// TwinCAT 3 PLC project Anker_Modenapark
// ProgramVersion: 3.1.4023.0
// libraries:
//   EfficientIO Communicator, * (EfficientIO)
//   Lynus Energy Basic, * (Lynus AG)
//   Lynus Persistent Data V1, * (Lynus AG)
//   Lynus Standards, * (Lynus AG)
//   Tc2_BABasic, * (Beckhoff Automation GmbH)
//   Tc2_Standard, * (Beckhoff Automation GmbH)
//   Tc2_System, * (Beckhoff Automation GmbH)
//   Tc2_Utilities, * (Beckhoff Automation GmbH)
//   Tc3_IotBase, * (Beckhoff Automation GmbH)
//   Tc3_JsonXml, * (Beckhoff Automation GmbH)
//   Tc3_Module, * (Beckhoff Automation GmbH)
// project tree:
//   / FastTask.TcTTO (not stored), MiddleTask.TcTTO, SlowTask.TcTTO
//   FBs/ FB_Shelly_Pro1PM.TcPOU, FB_Shelly_Pro1PM_Helper.TcPOU, FB_Shelly_Pro1PM_Helper_1.TcPOU (excluded from build), FB_Shelly_Pro1PM_Helper_2.TcPOU (excluded from build), FB_Shelly_Pro1PM_Helper_3.TcPOU (excluded from build), FB_TimeSwitch.TcPOU (not stored), FB_TimeSwitch_V2.TcPOU (not stored)
//   POUs/ prg5532EMS.TcPOU, prg5532Con.TcPOU, prgComEffIO.TcPOU, prg5532Grid.TcPOU, prgPersistent.TcPOU, prgRWEffIO.TcPOU, prgVarEffIO.TcPOU (not stored), prg_SystemTime.TcPOU (not stored)
// real-time tasks:
//   TASK FastTask: cycle T#5ms, priority 19, ADS port 350
//   TASK MiddleTask: cycle T#10ms, priority 20, ADS port 351
//   TASK SlowTask: cycle T#20ms, priority 21, ADS port 352
// I/O:
//   DEVICE Device 1 (Beckhoff CCAT)
//   DEVICE Device 2 (CX-BK)
//     Box 1 (CX-BK)
// variable links:
//   Anker_Modenapark/Anker_Modenapark Instance <-> Device 2 (CX-BK)/Box 1 (CX-BK)
//     MiddleTask Inputs/prg5532Grid.fbGrid.fbKL3403.byStateCH1 <-> Term 3 (KL3403)/Channel 1/State
//     MiddleTask Inputs/prg5532Grid.fbGrid.fbKL3403.byStateCH2 <-> Term 3 (KL3403)/Channel 2/State
//     MiddleTask Inputs/prg5532Grid.fbGrid.fbKL3403.byStateCH3 <-> Term 3 (KL3403)/Channel 3/State
//     MiddleTask Inputs/prg5532Grid.fbGrid.fbKL3403.iDataInCH1 <-> Term 3 (KL3403)/Channel 1/Data In
//     MiddleTask Inputs/prg5532Grid.fbGrid.fbKL3403.iDataInCH2 <-> Term 3 (KL3403)/Channel 2/Data In
//     MiddleTask Inputs/prg5532Grid.fbGrid.fbKL3403.iDataInCH3 <-> Term 3 (KL3403)/Channel 3/Data In
//     MiddleTask Inputs/prg5532Grid.fbKBusState.uiKBusState_OUT <-> Inputs/State
//     MiddleTask Outputs/prg5532EMS.bQ1Switch <-> Term 2 (KL2408)/Channel 1/Output
//     MiddleTask Outputs/prg5532Grid.fbGrid.fbKL3403.byCntrCH1 <-> Term 3 (KL3403)/Channel 1/Ctrl
//     MiddleTask Outputs/prg5532Grid.fbGrid.fbKL3403.byCntrCH2 <-> Term 3 (KL3403)/Channel 2/Ctrl
//     MiddleTask Outputs/prg5532Grid.fbGrid.fbKL3403.byCntrCH3 <-> Term 3 (KL3403)/Channel 3/Ctrl

CONFIGURATION Anker_Modenapark
    RESOURCE PLC ON TwinCAT3
        TASK MiddleTask(INTERVAL := T#10ms, PRIORITY := 20);
        TASK SlowTask(INTERVAL := T#20ms, PRIORITY := 21);
        PROGRAM prgPersistent WITH MiddleTask : prgPersistent;
        PROGRAM prg5532Grid WITH MiddleTask : prg5532Grid;
        PROGRAM prg5532Con WITH MiddleTask : prg5532Con;
        PROGRAM prg5532EMS WITH MiddleTask : prg5532EMS;
        PROGRAM prgComEffIO WITH SlowTask : prgComEffIO;
    END_RESOURCE
END_CONFIGURATION

// ---- POUs/prgPersistent.TcPOU
PROGRAM prgPersistent
VAR
	fbUSV		: FB_WritePersistentData_CX81xx;
END_VAR

fbUSV(
	eSaveModeData:= eUSVSaveMode.eSaveWhenPowerfail, 
	bLoadPersistentDataOk=> , 
	bPowerFailDetect=> , 
	bError=> , 
	bySaveProcess=> , 
	dwStorageLast24h=> , 
	udiErrorCode=> );

END_PROGRAM

// ---- POUs/prg5532Grid.TcPOU
PROGRAM prg5532Grid
VAR
	fbKBusState		: FB_K_Bus_State;
	fbGrid			: FB_EM_Beckhoff_KL3403;
	lrPowerGrid		: LREAL;							//{#lynus.ag#()}
	lrCounterGrid	: LREAL;							//{#lynus.ag#()}
	lrVoltageGridL1	: LREAL;							//{#lynus.ag#()}
	lrVoltageGridL2	: LREAL;							//{#lynus.ag#()}
	lrVoltageGridL3	: LREAL;							//{#lynus.ag#()}
	uint_BusState	: UINT;								//{#lynus.ag#()}
	int_LiveCount:int;
END_VAR

//The mapping of this function must be linked with the K-Bus State in the E/A Part
fbKBusState(	uiKBusState_OUT=> , 
				b_Kbus_notOk=> , 
				word_ErrorCount=> );
				
//The mapping of this function must be linked with the KL3403 in the E/A Part
fbGrid(
	bEnable:= TRUE, 
	bChannel1Invers:= TRUE,					//Invert power data when transformer are mounted upside down
	bChannel2Invers:= TRUE,
	bChannel3Invers:= TRUE,
	uiCurrentTransformerRatioL1:= 400, 		//Transformer ratio on the secondary side
	uiCurrentTransformerRatioL2:= 400, 
	uiCurrentTransformerRatioL3:= 400, 
	uiKBusState_IN:= fbKBusState.uiKBusState_OUT, 
	stDataEMPower=> , 
	stDataEMCounter=> , 
	stDataEMPowerRealTime=> , 
	stDataEMCounterRealTime=> , 
	diNrOfEM_OUT=> );

lrPowerGrid := fbGrid.stDataEMPower.lrPowerTotal;
	lrCounterGrid := fbGrid.stDataEMCounter.lrTotalCounterEnergy_Consumption;
		lrVoltageGridL1 := fbGrid.stDataEMPowerRealTime.lrVoltageL1N;
				lrVoltageGridL2 := fbGrid.stDataEMPowerRealTime.lrVoltageL2N;
					lrVoltageGridL3 := fbGrid.stDataEMPowerRealTime.lrVoltageL3N;


uint_BusState := fbKbusState.uiKBusState_OUT;
int_LiveCount:=int_LiveCount+1;

END_PROGRAM

// ---- POUs/prg5532Con.TcPOU
PROGRAM prg5532Con
VAR
	// Shelly1: 
//	fbShelly1				:	FB_Shelly_Pro1PM;
	lrS1P1Power				:	LREAL;			//{#lynus.ag#()}
	lrS1P1Power_kW			:	LREAL;			//{#lynus.ag#()}
	lrS1P1Voltage			:	LREAL;			//{#lynus.ag#()}
	lrS1P1Energy			:	LREAL;			//{#lynus.ag#()}
	lrS1P1Temperature		:	LREAL;			//{#lynus.ag#()}
	bS1P1On					:	BOOL;			//{#lynus.ag#()}
	bS1P1Off				:	BOOL;			//{#lynus.ag#()}
	bS1P1Switch				:	BOOL;			//{#lynus.ag#()}
	
	// Shelly2: 
//	fbShelly2				:	FB_Shelly_Pro1PM;
	lrS2P1Power				:	LREAL;			//{#lynus.ag#()}
	lrS2P1Power_kW			:	LREAL;			//{#lynus.ag#()}
	lrS2P1Voltage			:	LREAL;			//{#lynus.ag#()}
	lrS2P1Energy			:	LREAL;			//{#lynus.ag#()}
	lrS2P1Temperature		:	LREAL;			//{#lynus.ag#()}
	bS2P1On					:	BOOL;			//{#lynus.ag#()}
	bS2P1Off				:	BOOL;			//{#lynus.ag#()}
	bS2P1Switch				:	BOOL;			//{#lynus.ag#()}
	
	// Shelly3: 
//	fbShelly3				:	FB_Shelly_Pro1PM;
	lrS3P1Power				:	LREAL;			//{#lynus.ag#()}
	lrS3P1Power_kW			:	LREAL;			//{#lynus.ag#()}
	lrS3P1Voltage			:	LREAL;			//{#lynus.ag#()}
	lrS3P1Energy			:	LREAL;			//{#lynus.ag#()}
	lrS3P1Temperature		:	LREAL;			//{#lynus.ag#()}
	bS3P1On					:	BOOL;			//{#lynus.ag#()}
	bS3P1Off				:	BOOL;			//{#lynus.ag#()}
	bS3P1Switch				:	BOOL;			//{#lynus.ag#()}
	
	// Shelly4: 
//	fbShelly4				:	FB_Shelly_Pro1PM;
	lrS4P1Power				:	LREAL;			//{#lynus.ag#()}
	lrS4P1Power_kW			:	LREAL;			//{#lynus.ag#()}
	lrS4P1Voltage			:	LREAL;			//{#lynus.ag#()}
	lrS4P1Energy			:	LREAL;			//{#lynus.ag#()}
	lrS4P1Temperature		:	LREAL;			//{#lynus.ag#()}
	bS4P1On					:	BOOL;			//{#lynus.ag#()}
	bS4P1Off				:	BOOL;			//{#lynus.ag#()}
	bS4P1Switch				:	BOOL;			//{#lynus.ag#()}
	
	// Shelly5: 
//	fbShelly5				:	FB_Shelly_Pro1PM;
	lrS5P1Power				:	LREAL;			//{#lynus.ag#()}
	lrS5P1Power_kW			:	LREAL;			//{#lynus.ag#()}
	lrS5P1Voltage			:	LREAL;			//{#lynus.ag#()}
	lrS5P1Energy			:	LREAL;			//{#lynus.ag#()}
	lrS5P1Temperature		:	LREAL;			//{#lynus.ag#()}
	bS5P1On					:	BOOL;			//{#lynus.ag#()}
	bS5P1Off				:	BOOL;			//{#lynus.ag#()}
	bS5P1Switch				:	BOOL;			//{#lynus.ag#()}
	
	// Other
	lrRemainPower_kW		:	LREAL;			//{#lynus.ag#()}
	// state maschine for GET requests
	str_Array_IPs			: array[1..30] of STRING(15);			//arrays for IPs
	int_State: INT;
	
	int_Multiplier_1 			:INT:=1;								// multilpier received values, =2 when external fuse is on, was at the beginning
	int_Multiplier_2			:INT:=1;								// multilpier received values, =2 when external fuse is on, was at the beginning
	int_Multiplier_3 			:INT:=2;								// multilpier received values, =2 when external fuse is on, was at the beginning
	int_Multiplier_4 			:INT:=2;								// multilpier received values, =2 when external fuse is on, was at the beginning
	int_Multiplier_5 			:INT:=1;								// multilpier received values, =2 when external fuse is on, was at the beginning
	int_TimeoutCounter: ARRAY[1..30] OF INT;	
	int_SuccessCounter: ARRAY[1..30] OF INT;	
	int_ErrorCounter: ARRAY[1..30] OF INT;
	ton_wait: Ton;
	fbShelly				:	ARRAY[1..20] OF FB_Shelly_Pro1PM;
	f_Trig_Busy				:	ARRAY[1..20] OF f_trig;
	m_Error_HTTP: BOOL;							//{#lynus.ag#()}

	mTest: BOOL;
END_VAR

CASE int_State OF
	0: 		// Init State
	
	// define IPs
	str_Array_IPs[1]	:='10.55.32.131';
	str_Array_IPs[2]	:='10.55.32.132';
	str_Array_IPs[3]	:='10.55.32.133';			// bypass aktiv
	str_Array_IPs[4]	:='10.55.32.134';			// bypass aktiv    Getränkekühler RedBull
	str_Array_IPs[5]	:='10.55.32.135';
	str_Array_IPs[6]	:='';
	str_Array_IPs[7]	:='';
	str_Array_IPs[8]	:='';
	str_Array_IPs[9]	:='';
	str_Array_IPs[10]	:='';
	str_Array_IPs[11]	:='';
	str_Array_IPs[12]	:='';
	str_Array_IPs[13]	:='';
	str_Array_IPs[14]	:='';
	fbShelly[1].sHostname:= str_Array_IPs[1];
	fbShelly[2].sHostname:= str_Array_IPs[2];
	fbShelly[3].sHostname:= str_Array_IPs[3];
	fbShelly[4].sHostname:= str_Array_IPs[4];
	fbShelly[5].sHostname:= str_Array_IPs[5];
 
	
	// =2 for the beginning when bypass fuse is on
	int_Multiplier_1:=1;
	int_Multiplier_2:=1;
	int_Multiplier_3:=2;
	int_Multiplier_4:=2;
	int_Multiplier_5:=1;
	
	IF str_Array_IPs[1] <> '' THEN
		int_State :=1;
	END_IF
		
	1: 		// request
	
		fbShelly[int_State].bStart:= TRUE;
		fbShelly[int_State].bOnP1:= bS1P1On;
		fbShelly[int_State].bOffP1:= bS1P1Off;
	
		f_Trig_Busy[int_State](CLK :=fbShelly[int_State].bBusy);
			
		// go to next state
		IF f_Trig_Busy[int_State].Q  AND NOT fbShelly[int_State].bError THEN	
			int_SuccessCounter[int_State]	:= int_SuccessCounter[int_State]+1;
			lrS1P1Power 	:= 	fbShelly[int_State].lrpowerP1 * int_Multiplier_1;
			lrS1P1Energy 	:= 	fbShelly[int_State].lrenergyP1 * int_Multiplier_1;
			lrS1P1Voltage	:=	fbShelly[int_State].lrvoltageP1; 
			lrS1P1Temperature :=fbShelly[int_State].lrTemperatureP1;
			bS1P1Switch		:=	fbShelly[int_State].bStateP1;
		ELSIF  f_Trig_Busy[int_State].Q  AND fbShelly[int_State].bError THEN
			int_ErrorCounter[int_State]	:= int_ErrorCounter[int_State]+1;
		END_IF
		IF 	int_state < 20 AND str_Array_IPs[int_State+1] <> '' AND f_Trig_Busy[int_State].Q  THEN	
			fbShelly[int_State].bStart		:= FALSE;
			int_State := int_State+1;
		ELSIF  (str_Array_IPs[int_State+1] = '' OR int_state > 20) AND f_Trig_Busy[int_State].Q THEN
			fbShelly[int_State].bStart		:= FALSE;
			int_State := 100;			// wait state for new run
		END_IF		
	
	2: 		// request
	
		fbShelly[int_State].bStart:= TRUE;
		fbShelly[int_State].bOnP1:= bS2P1On;
		fbShelly[int_State].bOffP1:= bS2P1Off;
	
		f_Trig_Busy[int_State](CLK :=fbShelly[int_State].bBusy);
			
		// go to next state
		IF f_Trig_Busy[int_State].Q  AND NOT fbShelly[int_State].bError THEN	
			int_SuccessCounter[int_State]	:= int_SuccessCounter[int_State]+1;
			lrS2P1Power 	:= 	fbShelly[int_State].lrpowerP1 * int_Multiplier_2;
			lrS2P1Energy 	:= 	fbShelly[int_State].lrenergyP1 * int_Multiplier_2;
			lrS2P1Temperature :=fbShelly[int_State].lrTemperatureP1;
			lrS2P1Voltage	:=	fbShelly[int_State].lrvoltageP1; 
			bS2P1Switch		:=	fbShelly[int_State].bStateP1;
		ELSIF  f_Trig_Busy[int_State].Q  AND fbShelly[int_State].bError THEN
			int_ErrorCounter[int_State]	:= int_ErrorCounter[int_State]+1;
		END_IF
		IF 	int_state < 20 AND str_Array_IPs[int_State+1] <> '' AND f_Trig_Busy[int_State].Q  THEN	
			fbShelly[int_State].bStart		:= FALSE;
			int_State := int_State+1;
		ELSIF  (str_Array_IPs[int_State+1] = '' OR int_state > 20) AND f_Trig_Busy[int_State].Q THEN
			fbShelly[int_State].bStart		:= FALSE;
			int_State := 100;			// wait state for new run
		END_IF	
		
	3: 		// request
		fbShelly[int_State].bStart:= TRUE;
		fbShelly[int_State].bOnP1:= bS3P1On;
		fbShelly[int_State].bOffP1:= bS3P1Off;
	
		f_Trig_Busy[int_State](CLK :=fbShelly[int_State].bBusy);
			
		// go to next state
		IF f_Trig_Busy[int_State].Q  AND NOT fbShelly[int_State].bError THEN	
			int_SuccessCounter[int_State]	:= int_SuccessCounter[int_State]+1;
			lrS3P1Power 	:= 	fbShelly[int_State].lrpowerP1 * int_Multiplier_3;
			lrS3P1Energy 	:= 	fbShelly[int_State].lrenergyP1 * int_Multiplier_3;
			lrS3P1Temperature :=fbShelly[int_State].lrTemperatureP1;
			lrS3P1Voltage	:=	fbShelly[int_State].lrvoltageP1; 
			bS3P1Switch		:=	fbShelly[int_State].bStateP1;
		ELSIF  f_Trig_Busy[int_State].Q  AND fbShelly[int_State].bError THEN
			int_ErrorCounter[int_State]	:= int_ErrorCounter[int_State]+1;
		END_IF
		IF 	int_state < 20 AND str_Array_IPs[int_State+1] <> '' AND f_Trig_Busy[int_State].Q  THEN	
			fbShelly[int_State].bStart		:= FALSE;
			int_State := int_State+1;
		ELSIF  (str_Array_IPs[int_State+1] = '' OR int_state > 20) AND f_Trig_Busy[int_State].Q THEN
			fbShelly[int_State].bStart		:= FALSE;
			int_State := 100;			// wait state for new run
		END_IF	
	4: 		// request
	
		fbShelly[int_State].bStart:= TRUE;
		fbShelly[int_State].bOnP1:= bS4P1On;
		fbShelly[int_State].bOffP1:= bS4P1Off;
	
		f_Trig_Busy[int_State](CLK :=fbShelly[int_State].bBusy);
		IF f_Trig_Busy[int_State].Q THEN
			mTest:=TRUE;
		END_IF	
		// go to next state
		IF f_Trig_Busy[int_State].Q  AND NOT fbShelly[int_State].bError THEN	
			int_SuccessCounter[int_State]	:= int_SuccessCounter[int_State]+1;
			lrS4P1Power 	:= 	fbShelly[int_State].lrpowerP1 * int_Multiplier_4;
			lrS4P1Energy 	:= 	fbShelly[int_State].lrenergyP1 * int_Multiplier_4;
			lrS4P1Temperature :=fbShelly[int_State].lrTemperatureP1;
			lrS4P1Voltage	:=	fbShelly[int_State].lrvoltageP1; 
			bS4P1Switch		:=	fbShelly[int_State].bStateP1;
		ELSIF  f_Trig_Busy[int_State].Q  AND fbShelly[int_State].bError THEN
			int_ErrorCounter[int_State]	:= int_ErrorCounter[int_State]+1;
		END_IF
		IF 	int_state < 20 AND str_Array_IPs[int_State+1] <> '' AND f_Trig_Busy[int_State].Q  THEN	
			fbShelly[int_State].bStart		:= FALSE;
			int_State := int_State+1;
		ELSIF  (str_Array_IPs[int_State+1] = '' OR int_state > 20) AND f_Trig_Busy[int_State].Q THEN
			fbShelly[int_State].bStart		:= FALSE;
			int_State := 100;			// wait state for new run
		END_IF
		
	5: 		// request
	
		fbShelly[int_State].bStart:= TRUE;
		fbShelly[int_State].bOnP1:= bS5P1On;
		fbShelly[int_State].bOffP1:= bS5P1Off;
	
		f_Trig_Busy[int_State](CLK :=fbShelly[int_State].bBusy);
			
		// go to next state
		IF f_Trig_Busy[int_State].Q  AND NOT fbShelly[int_State].bError THEN	
			int_SuccessCounter[int_State]	:= int_SuccessCounter[int_State]+1;
			lrS5P1Power 	:= 	fbShelly[int_State].lrpowerP1 * int_Multiplier_5;
			lrS5P1Energy 	:= 	fbShelly[int_State].lrenergyP1 * int_Multiplier_5;
			lrS5P1Temperature :=fbShelly[int_State].lrTemperatureP1;
			lrS5P1Voltage	:=	fbShelly[int_State].lrvoltageP1; 
			bS5P1Switch		:=	fbShelly[int_State].bStateP1;
		ELSIF  f_Trig_Busy[int_State].Q  AND fbShelly[int_State].bError THEN
			int_ErrorCounter[int_State]	:= int_ErrorCounter[int_State]+1;
		END_IF
		IF 	int_state < 20 AND str_Array_IPs[int_State+1] <> '' AND f_Trig_Busy[int_State].Q  THEN	
			fbShelly[int_State].bStart		:= FALSE;
			int_State := int_State+1;
		ELSIF  (str_Array_IPs[int_State+1] = '' OR int_state > 20) AND f_Trig_Busy[int_State].Q THEN
			fbShelly[int_State].bStart		:= FALSE;
			int_State := 100;			// wait state for new run
		END_IF	
	
	100:		// wait state
	ton_wait.IN :=TRUE;
	IF ton_wait.Q THEN
		ton_wait.IN :=FALSE;
//		IF NOT fbShelly[1].bError THEN
			int_State := 1;			//// <-- must be 1
//		ELSIF fbShelly[1].bError AND prg_SystemTime.structSystemTime.wHour=4 AND prg_SystemTime.structSystemTime.wMinute>45 THEN
//			int_State := 1;
//		ELSE
//			int_State := 3;
//		END_IF
	END_IF		
END_CASE


// Shelly communication

fbShelly[1](tDelayRequest:= T#0S, );
fbShelly[2](tDelayRequest:= T#0S, );
fbShelly[3](tDelayRequest:= T#0S, );
fbShelly[4](tDelayRequest:= T#0S, );
fbShelly[5](tDelayRequest:= T#0S, );


// wait
ton_wait(PT:=T#3S);


// re-calc to kW
lrS1P1Power_kW := lrS1P1Power / 1000;
	lrS2P1Power_kW := lrS2P1Power / 1000;
		lrS3P1Power_kW := lrS3P1Power / 1000;
			lrS4P1Power_kW := lrS4P1Power / 1000;
				lrS5P1Power_kW := lrS5P1Power / 1000;
				
// Other
lrRemainPower_kW := LIMIT(0, prg5532Grid.lrPowerGrid - (lrS1P1Power_kW + lrS2P1Power_kW + lrS3P1Power_kW + lrS4P1Power_kW + lrS5P1Power_kW), 999999);
	
// on / off commands from EMS

// AC Shelly 1
fbShelly[1].bEnableControl := TRUE;		// prg5532EMS.FB_TimeSwitch_AC.b_Enable;
IF prg5532EMS.FB_TimeSwitch_AC.b_Output_On AND NOT fbShelly[1].bStateP1 THEN
	bS1P1On :=TRUE;
ELSE
	bS1P1On := FALSE;
END_IF
IF NOT prg5532EMS.FB_TimeSwitch_AC.b_Output_On AND fbShelly[1].bStateP1 THEN
	bS1P1Off :=TRUE;
ELSE
	bS1P1Off := FALSE;
END_IF
// Snackvitrine Shelly 2
fbShelly[2].bEnableControl := TRUE;		// prg5532EMS.FB_TimeSwitch_Snack.b_Enable;
IF prg5532EMS.FB_TimeSwitch_Snack.b_Output_On AND NOT fbShelly[2].bStateP1 THEN
	bS2P1On :=TRUE;
ELSE
	bS2P1On := FALSE;
END_IF
IF NOT prg5532EMS.FB_TimeSwitch_Snack.b_Output_On AND fbShelly[2].bStateP1 THEN
	bS2P1Off :=TRUE;
ELSE
	bS2P1Off := FALSE;
END_IF

// Außenbeleuchtung Shelly 5
fbShelly[5].bEnableControl := TRUE;		// prg5532EMS.FB_TimeSwitch_Outside.b_Enable;
IF prg5532EMS.RS_Outsidelight.Q1 AND NOT fbShelly[5].bStateP1 THEN
	bS5P1On :=TRUE;
ELSE
	bS5P1On := FALSE;
END_IF
IF NOT prg5532EMS.RS_Outsidelight.Q1 AND fbShelly[5].bStateP1 THEN
	bS5P1Off :=TRUE;
ELSE
	bS5P1Off := FALSE;
END_IF

// error bit to cloud 

m_Error_HTTP := fbShelly[1].bError OR fbShelly[2].bError OR fbShelly[5].bError;

END_PROGRAM

// ---- FBs/FB_Shelly_Pro1PM.TcPOU
FUNCTION_BLOCK FB_Shelly_Pro1PM
VAR_INPUT
	bStart				: BOOL;
	tDelayRequest		: TIME;				//Timer for delay before start with the next read or write Request
	sHostname			: STRING(255);		//Hostname or IP Adress from the Server
	bOnP1				: BOOL;
	bOffP1				: BOOL;
	bEnableControl		: BOOL;
END_VAR

VAR_OUTPUT
	bValidResult				: BOOL;															//Valid Result received from Server
    bBusy						: BOOL;															//Function is Busy
    bError						: BOOL;															//Error sucess
	bDone						: BOOL;															//True after the decoding from the received Json File
	bConnected					: BOOL;															//Connection to the Server
	hrErrorCode       			: HRESULT;														//Error Result from Http Client
	lrpowerP1					: LREAL;														//Received Value
	lrvoltageP1					: LREAL;														//Received Value
	lrenergyP1					: LREAL;														//Received Value
	lrTemperatureP1				: LREAL;														//Received Value
	bStateP1					: BOOL;
END_VAR

VAR
	fbClient					: FB_IotHttpClient;
	fbHttpGet					: FB_Shelly_Pro1PM_Helper;
	timStartRequest				: TON;															//Timer to Start the Request
	FPStartRequest				: R_TRIG;														//Internal positive Edge
	FPDone						: R_TRIG;														//Internal positive Edge
	FNStart						: F_TRIG;														//Internal negative Edge
	SwitchOnP1					: R_TRIG;
	SwitchOffP1					: R_TRIG;
	rs_Switch_ON: Rs;
	rs_Switch_OFF: RS;
	x: INT;
END_VAR

bError := FALSE;
(*------------------------------------------------------------------------------------Configure HTTP Client------------------------------------------------------------------------------------------------------*)

fbClient.sHostName := sHostname;
fbClient.tConnectionTimeout := T#25S;

IF NOT fbClient.bConfigured THEN 
	fbClient.nHostPort:= 80;
	fbClient.bKeepAlive := TRUE;
	fbClient.tConnectionTimeout := T#25S;
END_IF


//Timer to start the Request
FPStartRequest(CLK:= bStart, Q=> );
timStartRequest(	IN:= fbClient.bConfigured AND bStart AND NOT timStartRequest.Q, 
					PT:= tDelayRequest, 
					Q=> , 
					ET=> );
IF ((timStartRequest.Q AND NOT bBusy) OR (FPStartRequest.Q AND NOT bBusy AND fbClient.bConfigured)) THEN 
	fbHttpGet.bSend := TRUE; 
	x:=x+1;
END_IF

				
//Http Get Function
fbHttpGet(
	lrapowerP1 => lrpowerP1, 
	lrvoltageP1 => lrvoltageP1, 
	lraenergyP1 => lrenergyP1,
	lrTemperatureP1 => lrTemperatureP1,
	bSend:= , 
	fbClient:= fbClient, 
	bBusy=> bBusy, 
	bError=> ,
	sContentS0=> ,
	bStateP1=>bStateP1 );


fbHttpGet.bSend := FALSE;

FPDone(CLK:= bDone, Q=> );

// zum testen ob dadurch die verbindung aufrechtbleibt nach dem schalten 
// --> error geht nicht mehr low!
// IF NOT bError  THEN
	fbClient.Execute();
// ELSE
//	fbClient.Disconnect();
// END_IF

//Error
IF fbHttpGet.bError OR fbClient.bError THEN bError := TRUE; ELSE bError := FALSE; END_IF	
	hrErrorCode := fbClient.hrErrorCode;
	

// Relay Control, Switch P1
SwitchOnP1(CLK:=bOnP1);
rs_Switch_ON(	Set:= SwitchOnP1.Q AND bEnableControl,
				Reset1 := bStateP1);	// OR fbHttpGet.timTimeoutSwitch.Q);
				
IF rs_Switch_ON.Q1 AND bEnableControl THEN
	fbHttpGet.bSetOnP1 := TRUE;
ELSE
	fbHttpGet.bSetOnP1 := FALSE;
END_IF

SwitchOffP1(CLK:=bOffP1);
rs_Switch_OFF(	Set:= SwitchOffP1.Q AND bEnableControl,
				Reset1 := NOT bStateP1);	// OR fbHttpGet.timTimeoutSwitch.Q);
				
IF rs_Switch_OFF.Q1 AND bEnableControl THEN
	fbHttpGet.bSetOffP1 := TRUE;
ELSE
	fbHttpGet.bSetOffP1 := FALSE;
END_IF

END_FUNCTION_BLOCK

// ---- FBs/FB_Shelly_Pro1PM_Helper.TcPOU
FUNCTION_BLOCK FB_Shelly_Pro1PM_Helper
VAR_INPUT
	bSend			: BOOL;
	bSetOnP1		: BOOL;
	bSetOffP1		: BOOL;
END_VAR

VAR_IN_OUT
	fbClient		: FB_IotHttpClient;
END_VAR

VAR_OUTPUT
	bBusy			: BOOL;
	bError			: BOOL;
	bStateP1		: BOOL;
	lrapowerP1		: LREAL;
	lrvoltageP1		: LREAL;
	lraenergyP1		: LREAL;
	lrTemperatureP1	: LREAL;
END_VAR

VAR
	fbRequestSwitch0	: FB_IotHttpRequest;
	fbRequestSwitch1	: FB_IotHttpRequest;
	RisingEdge			: R_TRIG;
	RisingEdgeSetOnP1	: R_TRIG;
	RisingEdgeSetOffP1	: R_TRIG;
	fbJson				: FB_JsonDomParser;
	nState				: UDINT;
	timTimeout			: TON;
	tTimeOut			: TIME := T#2S;
	timTimeoutSwitch	: TON;
	tTimeOutSwitch		: TIME := T#5S;
	bGetContentResult	: BOOL;
	sContentS0			: STRING(511);
	
	bGetJsonResult		: BOOL;
	jsonDoc				: SJsonValue;
	jsonVal				: SJsonValue;
	
	nReqCount			: UDINT;	
	nResCount			: UDINT;
	nValidResCount		: UDINT;
	nErrCount			: UDINT;
	
	fbRequest2         : FB_IotHttpRequest;
	fbRequest3         : FB_IotHttpRequest;
	fbHeader            : FB_IotHttpHeaderFieldMap;
	fbHeader2            : FB_IotHttpHeaderFieldMap;
	
	sRealm	:	STRING(511);
	sPassword :	STRING(511) := ':sh3lly4ankerio2$$';
	snonce	:	STRING(511);
	scnonce	:	STRING(511);
	shash	: STRING(511);
	bhash	: BOOL;
	
	aData	: STRING(511);
	a_ha1	: ARRAY[0..31] OF BYTE;
	str_ha1 : STRING(511);
	str_Toha1   : STRING(511);
	udint_length_string : UDINT;
	
	a_ha2	: ARRAY[0..31] OF BYTE;
	str_ha2 : STRING(511);
	str_Toha2   : STRING(511);
	
	a_response	: ARRAY[0..31] OF BYTE;
	str_response : STRING(511);
	str_Toresponse   : STRING(511);

	str_authorization	: STRING(2048);
	
	sfincontent	: STRING(511);
	int_CountOffWrite: INT;
	int_CountOnWrite: INT;
	str_URI : STRING(50);
	int_Mode: INT;
	ton_Timeout: Ton;
	b_Done: BOOL;
	nState_Old: UDINT;
	int_ErrorCount: INT;
END_VAR

//Timer for Timeout
timTimeout(IN:= (nState = 1 AND bBusy) OR (nState = nState_Old AND bBusy), PT:= tTimeOut, Q=> , ET=> );
	IF timTimeout.Q THEN 
		nState := 0;
		bBusy := FALSE;
		bStateP1 := FALSE;
		lrapowerP1 := 0;
		lrvoltageP1 := 0;
		lraenergyP1 := 0;
		lrTemperatureP1 := 0;		
	END_IF
IF nState<> nState_old THEN
	nState_old := nState;
END_IF	
(*timTimeoutSwitch(IN:= bSetOnP1 OR bSetOffP1, PT:= tTimeOut, Q=> , ET=> );
	IF timTimeoutSwitch.Q THEN 
		bSetOnP1 := FALSE;
		bSetOffP1 := FALSE;
	END_IF
*)
IF bError THEN
	int_ErrorCount := int_ErrorCount+1;
	bError := FALSE;
END_IF

RisingEdge(CLK:= bSend );
RisingEdgeSetOnP1(CLK:= bSetOnP1 );
RisingEdgeSetOffP1(CLK:= bSetOffP1 );

CASE nState OF
	0:	
		IF RisingEdge.Q THEN 
			IF bSetOnP1 AND NOT b_Done THEN 
				// switch on
				str_URI :='/rpc/Switch.Set?id=0&on=true';
				int_Mode := 1;
				b_Done := TRUE;
				bBusy:= TRUE;
				bError:= FALSE;
				nState:= 1;
			ELSIF bSetOffP1 AND NOT b_Done THEN
				// switch off
				str_URI :='/rpc/Switch.Set?id=0&on=false';
				int_Mode := 2;
				b_Done := TRUE;
				bBusy:= TRUE;
				bError:= FALSE;
				nState:= 1;
			ELSIF ((bSetOnP1 OR bSetOffP1) AND  b_Done) OR (NOT bSetOnP1 AND NOT bSetOffP1) THEN
				// read
				str_URI :='/rpc/Switch.GetStatus?id=0';
				int_Mode := 0;
				b_Done := FALSE;
				bBusy:= TRUE;
				bError:= FALSE;
				nState:= 1;
			END_IF
		END_IF
	1:
		IF
			fbRequestSwitch0.SendRequest(sUri:=str_URI, fbClient:=fbClient, eRequestType:=ETcIotHttpRequestType.HTTP_Get, 0, 0, 0) THEN
			nState:= 2;
			nReqCount:= nReqCount+1;
		END_IF
	
	2:
		IF NOT fbRequestSwitch0.bBusy THEN
			bError:= TRUE;
			IF NOT fbRequestSwitch0.bError THEN
				bGetContentResult:= fbRequestSwitch0.GetHeaderField(pValue:= ADR(sContentS0), 
														 nValueSize:= SIZEOF(sContentS0), sField := 'WWW-Authenticate');
				IF fbRequestSwitch0.nStatusCode = 401 THEN
					bGetJsonResult:= FALSE;
						sRealm := sContentS0;
						sRealm := DELETE(sRealm, FIND(sRealm, 'realm') + 7, 0);
						sRealm := DELETE(sRealm, LEN(sRealm), FIND(sRealm, '"'));
						
						snonce := sContentS0;
						snonce := DELETE(snonce, FIND(snonce, 'nonce') + 7, 0);
						snonce := DELETE(snonce, LEN(snonce), FIND(snonce, '"'));
						
						scnonce := 'YmawvYzT';
					
						aData := sRealm;
						
						str_Toha1:=concat('admin:', sRealm);
						str_Toha1:=concat(str_Toha1, sPassword);
		 
						udint_length_string:= len2(ADR(str_Toha1));
						F_GenerateHashValue(E_HashMode.HASH_SHA256,ADR(str_Toha1),udint_length_string,ADR(a_ha1),32);
						
							str_ha1:=concat(byte_to_hexstr(a_ha1[0],2,TRUE),byte_to_hexstr(a_ha1[1],2,TRUE));
							str_ha1:=concat(str_ha1,byte_to_hexstr(a_ha1[2],2,TRUE));
							str_ha1:=concat(str_ha1,byte_to_hexstr(a_ha1[3],2,TRUE));
							str_ha1:=concat(str_ha1,byte_to_hexstr(a_ha1[4],2,TRUE));
							str_ha1:=concat(str_ha1,byte_to_hexstr(a_ha1[5],2,TRUE));
							str_ha1:=concat(str_ha1,byte_to_hexstr(a_ha1[6],2,TRUE));
							str_ha1:=concat(str_ha1,byte_to_hexstr(a_ha1[7],2,TRUE));
							str_ha1:=concat(str_ha1,byte_to_hexstr(a_ha1[8],2,TRUE));
							str_ha1:=concat(str_ha1,byte_to_hexstr(a_ha1[9],2,TRUE));
							str_ha1:=concat(str_ha1,byte_to_hexstr(a_ha1[10],2,TRUE));
							str_ha1:=concat(str_ha1,byte_to_hexstr(a_ha1[11],2,TRUE));
							str_ha1:=concat(str_ha1,byte_to_hexstr(a_ha1[12],2,TRUE));
							str_ha1:=concat(str_ha1,byte_to_hexstr(a_ha1[13],2,TRUE));
							str_ha1:=concat(str_ha1,byte_to_hexstr(a_ha1[14],2,TRUE));
							str_ha1:=concat(str_ha1,byte_to_hexstr(a_ha1[15],2,TRUE));
							str_ha1:=concat(str_ha1,byte_to_hexstr(a_ha1[16],2,TRUE));
							str_ha1:=concat(str_ha1,byte_to_hexstr(a_ha1[17],2,TRUE));
							str_ha1:=concat(str_ha1,byte_to_hexstr(a_ha1[18],2,TRUE));
							str_ha1:=concat(str_ha1,byte_to_hexstr(a_ha1[19],2,TRUE));
							str_ha1:=concat(str_ha1,byte_to_hexstr(a_ha1[20],2,TRUE));
							str_ha1:=concat(str_ha1,byte_to_hexstr(a_ha1[21],2,TRUE));
							str_ha1:=concat(str_ha1,byte_to_hexstr(a_ha1[22],2,TRUE));
							str_ha1:=concat(str_ha1,byte_to_hexstr(a_ha1[23],2,TRUE));
							str_ha1:=concat(str_ha1,byte_to_hexstr(a_ha1[24],2,TRUE));
							str_ha1:=concat(str_ha1,byte_to_hexstr(a_ha1[25],2,TRUE));
							str_ha1:=concat(str_ha1,byte_to_hexstr(a_ha1[26],2,TRUE));
							str_ha1:=concat(str_ha1,byte_to_hexstr(a_ha1[27],2,TRUE));
							str_ha1:=concat(str_ha1,byte_to_hexstr(a_ha1[28],2,TRUE));
							str_ha1:=concat(str_ha1,byte_to_hexstr(a_ha1[29],2,TRUE));
							str_ha1:=concat(str_ha1,byte_to_hexstr(a_ha1[30],2,TRUE));
							str_ha1:=concat(str_ha1,byte_to_hexstr(a_ha1[31],2,TRUE));
						
						str_Toha2:= concat('GET:',str_URI);
				 
						udint_length_string:= len2(ADR(str_Toha2));
						F_GenerateHashValue(E_HashMode.HASH_SHA256,ADR(str_Toha2),udint_length_string,ADR(a_ha2),32);
						
							str_ha2:=concat(byte_to_hexstr(a_ha2[0],2,TRUE),byte_to_hexstr(a_ha2[1],2,TRUE));
							str_ha2:=concat(str_ha2,byte_to_hexstr(a_ha2[2],2,TRUE));
							str_ha2:=concat(str_ha2,byte_to_hexstr(a_ha2[3],2,TRUE));
							str_ha2:=concat(str_ha2,byte_to_hexstr(a_ha2[4],2,TRUE));
							str_ha2:=concat(str_ha2,byte_to_hexstr(a_ha2[5],2,TRUE));
							str_ha2:=concat(str_ha2,byte_to_hexstr(a_ha2[6],2,TRUE));
							str_ha2:=concat(str_ha2,byte_to_hexstr(a_ha2[7],2,TRUE));
							str_ha2:=concat(str_ha2,byte_to_hexstr(a_ha2[8],2,TRUE));
							str_ha2:=concat(str_ha2,byte_to_hexstr(a_ha2[9],2,TRUE));
							str_ha2:=concat(str_ha2,byte_to_hexstr(a_ha2[10],2,TRUE));
							str_ha2:=concat(str_ha2,byte_to_hexstr(a_ha2[11],2,TRUE));
							str_ha2:=concat(str_ha2,byte_to_hexstr(a_ha2[12],2,TRUE));
							str_ha2:=concat(str_ha2,byte_to_hexstr(a_ha2[13],2,TRUE));
							str_ha2:=concat(str_ha2,byte_to_hexstr(a_ha2[14],2,TRUE));
							str_ha2:=concat(str_ha2,byte_to_hexstr(a_ha2[15],2,TRUE));
							str_ha2:=concat(str_ha2,byte_to_hexstr(a_ha2[16],2,TRUE));
							str_ha2:=concat(str_ha2,byte_to_hexstr(a_ha2[17],2,TRUE));
							str_ha2:=concat(str_ha2,byte_to_hexstr(a_ha2[18],2,TRUE));
							str_ha2:=concat(str_ha2,byte_to_hexstr(a_ha2[19],2,TRUE));
							str_ha2:=concat(str_ha2,byte_to_hexstr(a_ha2[20],2,TRUE));
							str_ha2:=concat(str_ha2,byte_to_hexstr(a_ha2[21],2,TRUE));
							str_ha2:=concat(str_ha2,byte_to_hexstr(a_ha2[22],2,TRUE));
							str_ha2:=concat(str_ha2,byte_to_hexstr(a_ha2[23],2,TRUE));
							str_ha2:=concat(str_ha2,byte_to_hexstr(a_ha2[24],2,TRUE));
							str_ha2:=concat(str_ha2,byte_to_hexstr(a_ha2[25],2,TRUE));
							str_ha2:=concat(str_ha2,byte_to_hexstr(a_ha2[26],2,TRUE));
							str_ha2:=concat(str_ha2,byte_to_hexstr(a_ha2[27],2,TRUE));
							str_ha2:=concat(str_ha2,byte_to_hexstr(a_ha2[28],2,TRUE));
							str_ha2:=concat(str_ha2,byte_to_hexstr(a_ha2[29],2,TRUE));
							str_ha2:=concat(str_ha2,byte_to_hexstr(a_ha2[30],2,TRUE));
							str_ha2:=concat(str_ha2,byte_to_hexstr(a_ha2[31],2,TRUE));
							
						// <ha1> + ":" + <nonce> + ":" + <nc> + ":" + <cnonce> + ":" + "auth" + ":" + <ha2>
						
						str_Toresponse:=concat(str_ha1,':');
						str_Toresponse:=concat(str_Toresponse,snonce);
						str_Toresponse:=concat(str_Toresponse,':00000001:');
						str_Toresponse:=concat(str_Toresponse,scnonce);
						str_Toresponse:=concat(str_Toresponse,':');
						str_Toresponse:=concat(str_Toresponse,'auth:');
						str_Toresponse:=concat(str_Toresponse,str_ha2);
						
						udint_length_string:= len2(ADR(str_Toresponse));
						F_GenerateHashValue(E_HashMode.HASH_SHA256,ADR(str_Toresponse),udint_length_string,ADR(a_response),32);
						
							str_response:=concat(byte_to_hexstr(a_response[0],2,TRUE),byte_to_hexstr(a_response[1],2,TRUE));
							str_response:=concat(str_response,byte_to_hexstr(a_response[2],2,TRUE));
							str_response:=concat(str_response,byte_to_hexstr(a_response[3],2,TRUE));
							str_response:=concat(str_response,byte_to_hexstr(a_response[4],2,TRUE));
							str_response:=concat(str_response,byte_to_hexstr(a_response[5],2,TRUE));
							str_response:=concat(str_response,byte_to_hexstr(a_response[6],2,TRUE));
							str_response:=concat(str_response,byte_to_hexstr(a_response[7],2,TRUE));
							str_response:=concat(str_response,byte_to_hexstr(a_response[8],2,TRUE));
							str_response:=concat(str_response,byte_to_hexstr(a_response[9],2,TRUE));
							str_response:=concat(str_response,byte_to_hexstr(a_response[10],2,TRUE));
							str_response:=concat(str_response,byte_to_hexstr(a_response[11],2,TRUE));
							str_response:=concat(str_response,byte_to_hexstr(a_response[12],2,TRUE));
							str_response:=concat(str_response,byte_to_hexstr(a_response[13],2,TRUE));
							str_response:=concat(str_response,byte_to_hexstr(a_response[14],2,TRUE));
							str_response:=concat(str_response,byte_to_hexstr(a_response[15],2,TRUE));
							str_response:=concat(str_response,byte_to_hexstr(a_response[16],2,TRUE));
							str_response:=concat(str_response,byte_to_hexstr(a_response[17],2,TRUE));
							str_response:=concat(str_response,byte_to_hexstr(a_response[18],2,TRUE));
							str_response:=concat(str_response,byte_to_hexstr(a_response[19],2,TRUE));
							str_response:=concat(str_response,byte_to_hexstr(a_response[20],2,TRUE));
							str_response:=concat(str_response,byte_to_hexstr(a_response[21],2,TRUE));
							str_response:=concat(str_response,byte_to_hexstr(a_response[22],2,TRUE));
							str_response:=concat(str_response,byte_to_hexstr(a_response[23],2,TRUE));
							str_response:=concat(str_response,byte_to_hexstr(a_response[24],2,TRUE));
							str_response:=concat(str_response,byte_to_hexstr(a_response[25],2,TRUE));
							str_response:=concat(str_response,byte_to_hexstr(a_response[26],2,TRUE));
							str_response:=concat(str_response,byte_to_hexstr(a_response[27],2,TRUE));
							str_response:=concat(str_response,byte_to_hexstr(a_response[28],2,TRUE));
							str_response:=concat(str_response,byte_to_hexstr(a_response[29],2,TRUE));
							str_response:=concat(str_response,byte_to_hexstr(a_response[30],2,TRUE));
							str_response:=concat(str_response,byte_to_hexstr(a_response[31],2,TRUE));
							
						// "Digest username=\"admin\", realm=\"shellypro4pm-083af27cfbac\", nonce=\"63768368\", uri=\"/rpc/Switch.GetStatus?id=0\", algorithm=\"SHA-256\", qop=auth, nc=00000001, cnonce=\"oKOklSrS\", response=\"d1d59d1e015dee0a3acfc97b20a0fa0ff851b03d79ca00df59ce018a63041468\""
						
						str_authorization:=concat('Digest username="admin", realm="',sRealm);
						str_authorization:=concat(str_authorization,'", nonce="');
						str_authorization:=concat(str_authorization,snonce);
						str_authorization:=concat(str_authorization,'", algorithm="SHA-256", uri="');
						str_authorization:=concat(str_authorization,str_URI);
						str_authorization:=concat(str_authorization,'", qop=auth, nc=00000001, cnonce="');
						str_authorization:=concat(str_authorization,scnonce);
						str_authorization:=concat(str_authorization,'", response="');
						str_authorization:=concat(str_authorization,str_response);
						str_authorization:=concat(str_authorization,'"');
						
						fbHeader.AddField('Authorization', str_authorization, FALSE);
						IF fbRequest2.SendRequest(sUri:= str_URI, fbClient:= fbClient, eRequestType:= ETcIotHttpRequestType.HTTP_Get, 0, 0, fbHeader) THEN
							nState:= 3;
							bBusy:= TRUE;
							bError:= FALSE;
						END_IF
				END_IF
			END_IF
		END_IF
	
	3:
		IF NOT fbRequest2.bBusy THEN
			bError:= TRUE;
			IF int_Mode<>0 THEN
				bError:= FALSE;
			END_IF
			IF NOT fbRequest2.bError THEN		//AND int_Mode=0 				 
				bGetContentResult:= fbRequest2.GetContent(pContent:= ADR(sfincontent), nContentSize:= SIZEOF(sfincontent), bSetNullTermination:= TRUE);
	
				IF fbRequest2.nStatusCode >= 200 AND fbRequest2.nStatusCode < 300 THEN
					bGetJsonResult:= FALSE;
					jsonDoc:= fbRequest2.GetJsonDomContent(fbJson);
					IF jsonDoc <> 0 THEN
						bGetJsonResult:= TRUE;
						IF fbJson.HasMember(jsonDoc, 'output')  THEN
							jsonVal:= fbJson.FindMember(jsonDoc, 'output');
							nValidResCount:= nValidResCount+1;					
							IF fbJson.IsBool(jsonVal) AND (fbJson.GetBool(jsonVal)=TRUE OR fbJson.GetBool(jsonVal)=FALSE) THEN							
								bStateP1:= fbJson.GetBool(jsonVal);									
							END_IF
						END_IF
						IF fbJson.HasMember(jsonDoc, 'apower')  THEN
							jsonVal:= fbJson.FindMember(jsonDoc, 'apower');
							nValidResCount:= nValidResCount+1;
							IF fbJson.IsDouble(jsonVal) AND fbJson.GetDouble(jsonVal)> -3.402823E+38 AND fbJson.GetDouble(jsonVal)< 3.402823E+38 THEN							
								lrapowerP1:= fbJson.GetDouble(jsonVal);									
							END_IF
						END_IF
						IF fbJson.HasMember(jsonDoc, 'voltage')  THEN
							jsonVal:= fbJson.FindMember(jsonDoc, 'voltage');
							nValidResCount:= nValidResCount+1;					
							IF fbJson.IsDouble(jsonVal) AND fbJson.GetDouble(jsonVal)> -3.402823E+38 AND fbJson.GetDouble(jsonVal)< 3.402823E+38 THEN
								lrvoltageP1:= fbJson.GetDouble(jsonVal);									
							END_IF
						END_IF
						IF fbJson.HasMember(jsonDoc, 'temperature')  THEN
							jsonVal:= fbJson.FindMember(jsonDoc, 'temperature');
							 IF fbJson.HasMember(jsonVal, 'tC') AND fbJson.GetDouble(jsonVal)> -3.402823E+38 AND fbJson.GetDouble(jsonVal)< 3.402823E+38 THEN							
								jsonVal:= fbJson.FindMember(jsonVal, 'tC');
								nValidResCount:= nValidResCount+1;					
								IF fbJson.IsDouble(jsonVal) AND fbJson.GetDouble(jsonVal)> -3.402823E+38 AND fbJson.GetDouble(jsonVal)< 3.402823E+38 THEN
									lrTemperatureP1:= fbJson.GetDouble(jsonVal);									
								END_IF
							END_IF
						END_IF
						IF fbJson.HasMember(jsonDoc, 'aenergy')  THEN
							jsonVal:= fbJson.FindMember(jsonDoc, 'aenergy');
							IF fbJson.HasMember(jsonVal, 'total') AND fbJson.GetDouble(jsonVal)> -3.402823E+38 AND fbJson.GetDouble(jsonVal)< 3.402823E+38 THEN							
								jsonVal:= fbJson.FindMember(jsonVal, 'total');
								nValidResCount:= nValidResCount+1;
								IF fbJson.IsDouble(jsonVal) AND fbJson.GetDouble(jsonVal)> -3.402823E+38 AND fbJson.GetDouble(jsonVal)< 3.402823E+38 THEN
									lraenergyP1:= fbJson.GetDouble(jsonVal);
								END_IF
							bError:= FALSE;
							END_IF
						END_IF	
					nResCount:= nResCount+1;			
					END_IF
				END_IF
			END_IF
		nState:= 4;
//		bBusy:= FALSE;
			IF bError THEN
				nErrCount:= nErrCount+1;
			END_IF
		ELSE
			ton_Timeout.IN := TRUE;
			IF ton_Timeout.Q THEN
				nState:= 3;	
				ton_Timeout.IN := FALSE;
			END_IF
		END_IF
	
	
	4:
		ton_Timeout.IN := FALSE;
		nState:= 6;
		
	6:
		bBusy:= FALSE;
		nState:= 0;

	
END_CASE

ton_Timeout(PT := T#5S);

END_FUNCTION_BLOCK

// ---- POUs/prg5532EMS.TcPOU
PROGRAM prg5532EMS
VAR
	//coffee machine relay
	bQ1Switch	AT%Q*	: BOOL;								//{#lynus.ag#()}
	FB_TimeSwitch_Coffee: FB_TimeSwitch_V2;
	FB_TimeSwitch_AC: FB_TimeSwitch_V2;
	FB_TimeSwitch_Snack: FB_TimeSwitch_V2;
	FB_TimeSwitch_RedBull: FB_TimeSwitch_V2;
	FB_TimeSwitch_Outside: FB_TimeSwitch_V2;

	b_Coffee_Manual_On: BOOL;						//{#lynus.ag#()}
	b_Coffee_Manual_Off: BOOL;						//{#lynus.ag#()}
	b_AC_Manual_On: BOOL;							//{#lynus.ag#()}
	b_AC_Manual_Off: BOOL;							//{#lynus.ag#()}
	b_Snack_Manual_On: BOOL;						//{#lynus.ag#()}
	b_Snack_Manual_Off: BOOL;						//{#lynus.ag#()}
	b_Outside_Manual_On: BOOL;						//{#lynus.ag#()}
	b_Outside_Manual_Off: BOOL;						//{#lynus.ag#()}

	fbCalcSunriseSunset   		: FB_CalcSunriseSunset;
	todSunrise            		: TOD;
	todSunset             		: TOD;
	fb_GetTimeZoneInfo	:FB_GetTimeZoneInformation;
	b_firstCycle: BOOL;
	RS_Outsidelight: RS;
	r_trig_on: R_trig;
	r_trig_off: R_trig;
	b_Status_CoffeeMaschine: BOOL;					//{#lynus.ag#()}
END_VAR
VAR PERSISTENT
// opening hours	
	byte_MoFr_Open_Hour		:BYTE;								//{#lynus.ag#()}
	byte_MoFr_Open_Minute	:BYTE;								//{#lynus.ag#()}
	byte_MoFr_Close_Hour	:BYTE;								//{#lynus.ag#()}
	byte_MoFr_Close_Minute	:BYTE;								//{#lynus.ag#()}
	byte_Sa_Open_Hour		:BYTE;								//{#lynus.ag#()}
	byte_Sa_Open_Minute		:BYTE;								//{#lynus.ag#()}
	byte_Sa_Close_Hour		:BYTE;								//{#lynus.ag#()}
	byte_Sa_Close_Minute	:BYTE;								//{#lynus.ag#()}
	byte_So_Open_Hour		:BYTE;								//{#lynus.ag#()}
	byte_So_Open_Minute		:BYTE;								//{#lynus.ag#()}
	byte_So_Close_Hour		:BYTE;								//{#lynus.ag#()}
	byte_So_Close_Minute	:BYTE;								//{#lynus.ag#()}
	
// offset coffeemaschine in hours			
	b_Enable_Control_Coffee		:BOOL;								//{#lynus.ag#()}
	real_Coffee_Offset_Start	:REAL;								//{#lynus.ag#()}
	real_Coffee_Offset_Stop		:REAL;								//{#lynus.ag#()}

// offset AC in hours			
	b_Enable_Control_AC			:BOOL;								//{#lynus.ag#()}
	real_AC_Offset_Start		:REAL;								//{#lynus.ag#()}
	real_AC_Offset_Stop			:REAL;								//{#lynus.ag#()}
	
// offset snack in hours			
	b_Enable_Control_Snack		:BOOL;								//{#lynus.ag#()}
	real_Snack_Offset_Start		:REAL;								//{#lynus.ag#()}
	real_Snack_Offset_Stop		:REAL;								//{#lynus.ag#()}

// offset RedBull Cooler in hours			
	b_Enable_Control_RedBull	:BOOL;								//{#lynus.ag#()}
	real_RedBull_Offset_Start	:REAL;								//{#lynus.ag#()}
	real_RedBull_Offset_Stop	:REAL;								//{#lynus.ag#()}

// offset outside light in hours			
	b_Enable_Control_Outside	:BOOL;								//{#lynus.ag#()}
	real_Outside_Offset_Start	:REAL;								//{#lynus.ag#()}
	real_Outside_Offset_Stop	:REAL;								//{#lynus.ag#()}
END_VAR


FB_TimeSwitch_Coffee(
	b_Enable:= b_Enable_Control_Coffee, 
	b_StatusOn:= NOT bQ1Switch, 
	structSystemTime:=prg_SystemTime.structSystemTime , 
	byte_MoFr_Open_Hour:= byte_MoFr_Open_Hour , 
	byte_MoFr_Open_Minute:= byte_MoFr_Open_Minute, 
	byte_MoFr_Close_Hour:= byte_MoFr_Close_Hour , 
	byte_MoFr_Close_Minute:= byte_MoFr_Close_Minute, 
	byte_Sa_Open_Hour:= byte_Sa_Open_Hour, 
	byte_Sa_Open_Minute:= byte_Sa_Open_Minute , 
	byte_Sa_Close_Hour:= byte_Sa_Close_Hour , 
	byte_Sa_Close_Minute:= byte_Sa_Close_Minute, 
	byte_So_Open_Hour:= byte_So_Open_Hour, 
	byte_So_Open_Minute:= byte_So_Open_Minute, 
	byte_So_Close_Hour:= byte_So_Close_Hour, 
	byte_So_Close_Minute:= byte_So_Close_Minute, 
	real_Offset_Start:= real_Coffee_Offset_Start , 
	real_Offset_Stop:= real_Coffee_Offset_Stop , 
	b_On_Manual:= b_Coffee_Manual_On, 
	b_Off_Manual:= b_Coffee_Manual_Off, 
	b_Output_On=> , 
	b_Error=> );
IF NOT FB_TimeSwitch_Coffee.b_Output_On THEN
	bQ1Switch := TRUE;
ELSIF FB_TimeSwitch_Coffee.b_Output_On THEN
	bQ1Switch := FALSE;
END_IF
b_Status_CoffeeMaschine := NOT bQ1Switch;
	
FB_TimeSwitch_AC(
	b_Enable:= b_Enable_Control_AC, 
	b_StatusOn:= prg5532CON.fbShelly[1].bStateP1, 
	structSystemTime:= prg_SystemTime.structSystemTime , 
	byte_MoFr_Open_Hour:= byte_MoFr_Open_Hour , 
	byte_MoFr_Open_Minute:= byte_MoFr_Open_Minute, 
	byte_MoFr_Close_Hour:= byte_MoFr_Close_Hour , 
	byte_MoFr_Close_Minute:= byte_MoFr_Close_Minute, 
	byte_Sa_Open_Hour:= byte_Sa_Open_Hour, 
	byte_Sa_Open_Minute:= byte_Sa_Open_Minute , 
	byte_Sa_Close_Hour:= byte_Sa_Close_Hour , 
	byte_Sa_Close_Minute:= byte_Sa_Close_Minute, 
	byte_So_Open_Hour:= byte_So_Open_Hour, 
	byte_So_Open_Minute:= byte_So_Open_Minute, 
	byte_So_Close_Hour:= byte_So_Close_Hour, 
	byte_So_Close_Minute:= byte_So_Close_Minute, 
	real_Offset_Start:= real_AC_Offset_Start , 
	real_Offset_Stop:= real_AC_Offset_Stop , 
	b_On_Manual:= b_AC_Manual_On, 
	b_Off_Manual:= b_AC_Manual_Off, 
	b_Output_On=> , 
	b_Error=> );

FB_TimeSwitch_Snack(
	b_Enable:= b_Enable_Control_Snack, 
	b_StatusOn:= prg5532CON.fbShelly[2].bStateP1, 
	structSystemTime:= prg_SystemTime.structSystemTime , 
	byte_MoFr_Open_Hour:= byte_MoFr_Open_Hour , 
	byte_MoFr_Open_Minute:= byte_MoFr_Open_Minute, 
	byte_MoFr_Close_Hour:= byte_MoFr_Close_Hour , 
	byte_MoFr_Close_Minute:= byte_MoFr_Close_Minute, 
	byte_Sa_Open_Hour:= byte_Sa_Open_Hour, 
	byte_Sa_Open_Minute:= byte_Sa_Open_Minute , 
	byte_Sa_Close_Hour:= byte_Sa_Close_Hour , 
	byte_Sa_Close_Minute:= byte_Sa_Close_Minute, 
	byte_So_Open_Hour:= byte_So_Open_Hour, 
	byte_So_Open_Minute:= byte_So_Open_Minute, 
	byte_So_Close_Hour:= byte_So_Close_Hour, 
	byte_So_Close_Minute:= byte_So_Close_Minute, 
	real_Offset_Start:= real_Snack_Offset_Start , 
	real_Offset_Stop:= real_Snack_Offset_Stop , 
	b_On_Manual:= b_Snack_Manual_On, 
	b_Off_Manual:= b_Snack_Manual_Off, 
	b_Output_On=> , 
	b_Error=> );
	
FB_TimeSwitch_Outside(
	b_Enable:= b_Enable_Control_Outside, 
	b_StatusOn:= prg5532CON.fbShelly[5].bStateP1, 
	structSystemTime:= prg_SystemTime.structSystemTime , 
	byte_MoFr_Open_Hour:= byte_MoFr_Open_Hour , 
	byte_MoFr_Open_Minute:= byte_MoFr_Open_Minute, 
	byte_MoFr_Close_Hour:= byte_MoFr_Close_Hour , 
	byte_MoFr_Close_Minute:= byte_MoFr_Close_Minute, 
	byte_Sa_Open_Hour:= byte_Sa_Open_Hour, 
	byte_Sa_Open_Minute:= byte_Sa_Open_Minute , 
	byte_Sa_Close_Hour:= byte_Sa_Close_Hour , 
	byte_Sa_Close_Minute:= byte_Sa_Close_Minute, 
	byte_So_Open_Hour:= byte_So_Open_Hour, 
	byte_So_Open_Minute:= byte_So_Open_Minute, 
	byte_So_Close_Hour:= byte_So_Close_Hour, 
	byte_So_Close_Minute:= byte_So_Close_Minute, 
	real_Offset_Start:= real_Outside_Offset_Start , 
	real_Offset_Stop:= real_Outside_Offset_Stop , 
	b_On_Manual:= b_Outside_Manual_On, 
	b_Off_Manual:= b_Outside_Manual_Off, 
	b_Output_On=> , 
	b_Error=> );
	
// calculate sunset / sunrise
// find out the time details
fb_GetTimeZoneInfo(
	sNetID:= '', 
	bExecute:= prg_SystemTime.structSystemTime.wHour = 4 OR NOT b_firstCycle, 
	tTimeout:= T#5S, 
	bBusy=> , 
	bError=> , 
	nErrID=> , 
	tzID=> , 
	tzInfo=> );
b_firstCycle := TRUE;

fbCalcSunriseSunset(
	fDegreeOfLongitude := 16.3731,   (* Longitude of Vienna *)
	fDegreeOfLatitude := 48.2083,   (* Latitude of Vienna*)
	fReferenceMeridian := SEL( fb_GetTimeZoneInfo.tzID = eTimeZoneID_Daylight ,15,30),  (* Central European Time 15 Winter Timer / 30 Summer Time *)
	dCurrentDate := DT_TO_DATE(SYSTEMTIME_TO_Dt (prg_SystemTime.structSystemTime)),
	todSunrise => todSunrise,
	todSunset => todSunset);

r_trig_on (clk := FB_TimeSwitch_Outside.b_Output_On AND DT_TO_TOD(systemtime_to_dt(prg_SystemTime.structSystemTime))< (todSunrise +  T#1H) );
r_trig_off (clk := NOT FB_TimeSwitch_Outside.b_Output_On);

RS_Outsidelight(	Set := r_trig_on.Q OR ((todSunset - T#2H) =  DT_TO_TOD(systemtime_to_dt(prg_SystemTime.structSystemTime)) AND FB_TimeSwitch_Outside.b_Output_On) OR b_Outside_Manual_On ,
					Reset1 := r_trig_off.Q OR ((todSunrise +  T#1H)= DT_TO_TOD(systemtime_to_dt(prg_SystemTime.structSystemTime))) OR b_Outside_Manual_Off,
					Q1 => );

END_PROGRAM

// ---- POUs/prgComEffIO.TcPOU
PROGRAM prgComEffIO
VAR
	fbCom		: FB_MqttCommunicator;
END_VAR

fbCom(
	bConnect:= TRUE, 
	sUserName:= 'eb1d6961-5914-4eb4-a228-c95326bab078', 
	sUserPassword:= '385e050b-6c7d-4c72-ab76-b82697410544', 
	eSavePositionCertificate:= eSavePositionOnPLC.ePostionHardDisk, 
	bConnected=> , 
	bError=> , 
	hrErrorCode=> , 
	eConnectionState=> , 
	eErrorMessage_Out=> );

prg_SystemTime();

END_PROGRAM

// ---- FBs/FB_Shelly_Pro1PM_Helper_1.TcPOU
FUNCTION_BLOCK FB_Shelly_Pro1PM_Helper_1
VAR_INPUT
	bSend			: BOOL;
	bSetOnP1		: BOOL;
	bSetOffP1		: BOOL;
END_VAR

VAR_IN_OUT
	fbClient		: FB_IotHttpClient;
END_VAR

VAR_OUTPUT
	bBusy			: BOOL;
	bError			: BOOL;
	bStateP1		: BOOL;
	lrapowerP1		: LREAL;
	lrvoltageP1		: LREAL;
	lraenergyP1		: LREAL;
	lrTemperatureP1	: LREAL;
END_VAR

VAR
	fbRequestSwitch0	: FB_IotHttpRequest;
	RisingEdge			: R_TRIG;
	RisingEdgeSetOnP1	: R_TRIG;
	RisingEdgeSetOffP1	: R_TRIG;
	fbJson				: FB_JsonDomParser;
	nState				: UDINT;
	timTimeout			: TON;
	tTimeOut			: TIME := T#30S;
	timTimeoutSwitch	: TON;
	tTimeOutSwitch		: TIME := T#5S;
	bGetContentResult	: BOOL;
	sContentS0			: STRING(511);
	
	bGetJsonResult		: BOOL;
	jsonDoc				: SJsonValue;
	jsonVal				: SJsonValue;
	
	nReqCount			: UDINT;	
	nResCount			: UDINT;
	nValidResCount		: UDINT;
	nErrCount			: UDINT;
	
	fbRequest2         : FB_IotHttpRequest;
	fbHeader            : FB_IotHttpHeaderFieldMap;
	
	sRealm	:	STRING(511);
	sPassword :	STRING(511) := ':sh3lly4ankerio2$$';
	snonce	:	STRING(511);
	scnonce	:	STRING(511);
	shash	: STRING(511);
	bhash	: BOOL;
	
	aData	: STRING(511);
	a_ha1	: ARRAY[0..31] OF BYTE;
	str_ha1 : STRING(511);
	str_Toha1   : STRING(511);
	udint_length_string : UDINT;
	
	a_ha2	: ARRAY[0..31] OF BYTE;
	str_ha2 : STRING(511);
	str_Toha2   : STRING(511);
	
	a_response	: ARRAY[0..31] OF BYTE;
	str_response : STRING(511);
	str_Toresponse   : STRING(511);

	str_authorization	: STRING(2048);
	
	sfincontent	: STRING(511);
END_VAR

//Timer for Timeout
timTimeout(IN:= nState = 1 AND bBusy, PT:= tTimeOut, Q=> , ET=> );
	IF timTimeout.Q THEN 
		nState := 0;
		bBusy := FALSE;
	END_IF
	
timTimeoutSwitch(IN:= bSetOnP1 OR bSetOffP1, PT:= tTimeOut, Q=> , ET=> );
	IF timTimeoutSwitch.Q THEN 
		bSetOnP1 := FALSE;
		bSetOffP1 := FALSE;
	END_IF

RisingEdge(CLK:= bSend );
RisingEdgeSetOnP1(CLK:= bSetOnP1 );
RisingEdgeSetOffP1(CLK:= bSetOffP1 );

CASE nState OF
0:	
	IF RisingEdge.Q THEN 
		IF
			fbRequestSwitch0.SendRequest(sUri:='/rpc/Switch.GetStatus?id=0', fbClient:=fbClient, eRequestType:=ETcIotHttpRequestType.HTTP_Get, 0, 0, 0) THEN
			nState:= 1;
			nReqCount:= nReqCount+1;
			bBusy:= TRUE;
			bError:= FALSE;
		END_IF					
	END_IF
	
	IF RisingEdgeSetOnP1.Q THEN 
		IF
			fbRequestSwitch0.SendRequest(sUri:='/rpc/Switch.Set?id=0&on=true', fbClient:=fbClient, eRequestType:=ETcIotHttpRequestType.HTTP_Get, 0, 0, 0) THEN				
			bSetOnP1 := FALSE;
			nState:= 1;
			bBusy:= TRUE;
			bError:= FALSE;
		END_IF					
	END_IF
	
	IF RisingEdgeSetOffP1.Q THEN 
		IF
			fbRequestSwitch0.SendRequest(sUri:='/rpc/Switch.Set?id=0&on=false', fbClient:=fbClient, eRequestType:=ETcIotHttpRequestType.HTTP_Get, 0, 0, 0) THEN				
			bSetOffP1 := FALSE;
			nState:= 1;
			bBusy:= TRUE;
			bError:= FALSE;
		END_IF					
	END_IF

1:
    IF NOT fbRequestSwitch0.bBusy THEN
        bError:= TRUE;
        IF NOT fbRequestSwitch0.bError THEN
            bGetContentResult:= fbRequestSwitch0.GetHeaderField(pValue:= ADR(sContentS0), 
                                                     nValueSize:= SIZEOF(sContentS0), sField := 'WWW-Authenticate');
            IF fbRequestSwitch0.nStatusCode = 401 THEN
                bGetJsonResult:= FALSE;
					sRealm := sContentS0;
                    sRealm := DELETE(sRealm, FIND(sRealm, 'realm') + 7, 0);
					sRealm := DELETE(sRealm, LEN(sRealm), FIND(sRealm, '"'));
					
					snonce := sContentS0;
					snonce := DELETE(snonce, FIND(snonce, 'nonce') + 7, 0);
					snonce := DELETE(snonce, LEN(snonce), FIND(snonce, '"'));
					
					scnonce := 'YmawvYzT';
				
					aData := sRealm;
					
					str_Toha1:=concat('admin:', sRealm);
    				str_Toha1:=concat(str_Toha1, sPassword);
     
   					udint_length_string:= len2(ADR(str_Toha1));
					F_GenerateHashValue(E_HashMode.HASH_SHA256,ADR(str_Toha1),udint_length_string,ADR(a_ha1),32);
					
						str_ha1:=concat(byte_to_hexstr(a_ha1[0],2,TRUE),byte_to_hexstr(a_ha1[1],2,TRUE));
						str_ha1:=concat(str_ha1,byte_to_hexstr(a_ha1[2],2,TRUE));
						str_ha1:=concat(str_ha1,byte_to_hexstr(a_ha1[3],2,TRUE));
						str_ha1:=concat(str_ha1,byte_to_hexstr(a_ha1[4],2,TRUE));
						str_ha1:=concat(str_ha1,byte_to_hexstr(a_ha1[5],2,TRUE));
						str_ha1:=concat(str_ha1,byte_to_hexstr(a_ha1[6],2,TRUE));
						str_ha1:=concat(str_ha1,byte_to_hexstr(a_ha1[7],2,TRUE));
						str_ha1:=concat(str_ha1,byte_to_hexstr(a_ha1[8],2,TRUE));
						str_ha1:=concat(str_ha1,byte_to_hexstr(a_ha1[9],2,TRUE));
						str_ha1:=concat(str_ha1,byte_to_hexstr(a_ha1[10],2,TRUE));
						str_ha1:=concat(str_ha1,byte_to_hexstr(a_ha1[11],2,TRUE));
						str_ha1:=concat(str_ha1,byte_to_hexstr(a_ha1[12],2,TRUE));
						str_ha1:=concat(str_ha1,byte_to_hexstr(a_ha1[13],2,TRUE));
						str_ha1:=concat(str_ha1,byte_to_hexstr(a_ha1[14],2,TRUE));
						str_ha1:=concat(str_ha1,byte_to_hexstr(a_ha1[15],2,TRUE));
						str_ha1:=concat(str_ha1,byte_to_hexstr(a_ha1[16],2,TRUE));
						str_ha1:=concat(str_ha1,byte_to_hexstr(a_ha1[17],2,TRUE));
						str_ha1:=concat(str_ha1,byte_to_hexstr(a_ha1[18],2,TRUE));
						str_ha1:=concat(str_ha1,byte_to_hexstr(a_ha1[19],2,TRUE));
						str_ha1:=concat(str_ha1,byte_to_hexstr(a_ha1[20],2,TRUE));
						str_ha1:=concat(str_ha1,byte_to_hexstr(a_ha1[21],2,TRUE));
						str_ha1:=concat(str_ha1,byte_to_hexstr(a_ha1[22],2,TRUE));
						str_ha1:=concat(str_ha1,byte_to_hexstr(a_ha1[23],2,TRUE));
						str_ha1:=concat(str_ha1,byte_to_hexstr(a_ha1[24],2,TRUE));
						str_ha1:=concat(str_ha1,byte_to_hexstr(a_ha1[25],2,TRUE));
						str_ha1:=concat(str_ha1,byte_to_hexstr(a_ha1[26],2,TRUE));
						str_ha1:=concat(str_ha1,byte_to_hexstr(a_ha1[27],2,TRUE));
						str_ha1:=concat(str_ha1,byte_to_hexstr(a_ha1[28],2,TRUE));
						str_ha1:=concat(str_ha1,byte_to_hexstr(a_ha1[29],2,TRUE));
						str_ha1:=concat(str_ha1,byte_to_hexstr(a_ha1[30],2,TRUE));
						str_ha1:=concat(str_ha1,byte_to_hexstr(a_ha1[31],2,TRUE));
					
					str_Toha2:='GET:/rpc/Switch.GetStatus?id=0';
     
   					udint_length_string:= len2(ADR(str_Toha2));
					F_GenerateHashValue(E_HashMode.HASH_SHA256,ADR(str_Toha2),udint_length_string,ADR(a_ha2),32);
					
						str_ha2:=concat(byte_to_hexstr(a_ha2[0],2,TRUE),byte_to_hexstr(a_ha2[1],2,TRUE));
						str_ha2:=concat(str_ha2,byte_to_hexstr(a_ha2[2],2,TRUE));
						str_ha2:=concat(str_ha2,byte_to_hexstr(a_ha2[3],2,TRUE));
						str_ha2:=concat(str_ha2,byte_to_hexstr(a_ha2[4],2,TRUE));
						str_ha2:=concat(str_ha2,byte_to_hexstr(a_ha2[5],2,TRUE));
						str_ha2:=concat(str_ha2,byte_to_hexstr(a_ha2[6],2,TRUE));
						str_ha2:=concat(str_ha2,byte_to_hexstr(a_ha2[7],2,TRUE));
						str_ha2:=concat(str_ha2,byte_to_hexstr(a_ha2[8],2,TRUE));
						str_ha2:=concat(str_ha2,byte_to_hexstr(a_ha2[9],2,TRUE));
						str_ha2:=concat(str_ha2,byte_to_hexstr(a_ha2[10],2,TRUE));
						str_ha2:=concat(str_ha2,byte_to_hexstr(a_ha2[11],2,TRUE));
						str_ha2:=concat(str_ha2,byte_to_hexstr(a_ha2[12],2,TRUE));
						str_ha2:=concat(str_ha2,byte_to_hexstr(a_ha2[13],2,TRUE));
						str_ha2:=concat(str_ha2,byte_to_hexstr(a_ha2[14],2,TRUE));
						str_ha2:=concat(str_ha2,byte_to_hexstr(a_ha2[15],2,TRUE));
						str_ha2:=concat(str_ha2,byte_to_hexstr(a_ha2[16],2,TRUE));
						str_ha2:=concat(str_ha2,byte_to_hexstr(a_ha2[17],2,TRUE));
						str_ha2:=concat(str_ha2,byte_to_hexstr(a_ha2[18],2,TRUE));
						str_ha2:=concat(str_ha2,byte_to_hexstr(a_ha2[19],2,TRUE));
						str_ha2:=concat(str_ha2,byte_to_hexstr(a_ha2[20],2,TRUE));
						str_ha2:=concat(str_ha2,byte_to_hexstr(a_ha2[21],2,TRUE));
						str_ha2:=concat(str_ha2,byte_to_hexstr(a_ha2[22],2,TRUE));
						str_ha2:=concat(str_ha2,byte_to_hexstr(a_ha2[23],2,TRUE));
						str_ha2:=concat(str_ha2,byte_to_hexstr(a_ha2[24],2,TRUE));
						str_ha2:=concat(str_ha2,byte_to_hexstr(a_ha2[25],2,TRUE));
						str_ha2:=concat(str_ha2,byte_to_hexstr(a_ha2[26],2,TRUE));
						str_ha2:=concat(str_ha2,byte_to_hexstr(a_ha2[27],2,TRUE));
						str_ha2:=concat(str_ha2,byte_to_hexstr(a_ha2[28],2,TRUE));
						str_ha2:=concat(str_ha2,byte_to_hexstr(a_ha2[29],2,TRUE));
						str_ha2:=concat(str_ha2,byte_to_hexstr(a_ha2[30],2,TRUE));
						str_ha2:=concat(str_ha2,byte_to_hexstr(a_ha2[31],2,TRUE));
						
					// <ha1> + ":" + <nonce> + ":" + <nc> + ":" + <cnonce> + ":" + "auth" + ":" + <ha2>
					
					str_Toresponse:=concat(str_ha1,':');
					str_Toresponse:=concat(str_Toresponse,snonce);
					str_Toresponse:=concat(str_Toresponse,':00000001:');
					str_Toresponse:=concat(str_Toresponse,scnonce);
					str_Toresponse:=concat(str_Toresponse,':');
					str_Toresponse:=concat(str_Toresponse,'auth:');
					str_Toresponse:=concat(str_Toresponse,str_ha2);
					
					udint_length_string:= len2(ADR(str_Toresponse));
					F_GenerateHashValue(E_HashMode.HASH_SHA256,ADR(str_Toresponse),udint_length_string,ADR(a_response),32);
					
						str_response:=concat(byte_to_hexstr(a_response[0],2,TRUE),byte_to_hexstr(a_response[1],2,TRUE));
						str_response:=concat(str_response,byte_to_hexstr(a_response[2],2,TRUE));
						str_response:=concat(str_response,byte_to_hexstr(a_response[3],2,TRUE));
						str_response:=concat(str_response,byte_to_hexstr(a_response[4],2,TRUE));
						str_response:=concat(str_response,byte_to_hexstr(a_response[5],2,TRUE));
						str_response:=concat(str_response,byte_to_hexstr(a_response[6],2,TRUE));
						str_response:=concat(str_response,byte_to_hexstr(a_response[7],2,TRUE));
						str_response:=concat(str_response,byte_to_hexstr(a_response[8],2,TRUE));
						str_response:=concat(str_response,byte_to_hexstr(a_response[9],2,TRUE));
						str_response:=concat(str_response,byte_to_hexstr(a_response[10],2,TRUE));
						str_response:=concat(str_response,byte_to_hexstr(a_response[11],2,TRUE));
						str_response:=concat(str_response,byte_to_hexstr(a_response[12],2,TRUE));
						str_response:=concat(str_response,byte_to_hexstr(a_response[13],2,TRUE));
						str_response:=concat(str_response,byte_to_hexstr(a_response[14],2,TRUE));
						str_response:=concat(str_response,byte_to_hexstr(a_response[15],2,TRUE));
						str_response:=concat(str_response,byte_to_hexstr(a_response[16],2,TRUE));
						str_response:=concat(str_response,byte_to_hexstr(a_response[17],2,TRUE));
						str_response:=concat(str_response,byte_to_hexstr(a_response[18],2,TRUE));
						str_response:=concat(str_response,byte_to_hexstr(a_response[19],2,TRUE));
						str_response:=concat(str_response,byte_to_hexstr(a_response[20],2,TRUE));
						str_response:=concat(str_response,byte_to_hexstr(a_response[21],2,TRUE));
						str_response:=concat(str_response,byte_to_hexstr(a_response[22],2,TRUE));
						str_response:=concat(str_response,byte_to_hexstr(a_response[23],2,TRUE));
						str_response:=concat(str_response,byte_to_hexstr(a_response[24],2,TRUE));
						str_response:=concat(str_response,byte_to_hexstr(a_response[25],2,TRUE));
						str_response:=concat(str_response,byte_to_hexstr(a_response[26],2,TRUE));
						str_response:=concat(str_response,byte_to_hexstr(a_response[27],2,TRUE));
						str_response:=concat(str_response,byte_to_hexstr(a_response[28],2,TRUE));
						str_response:=concat(str_response,byte_to_hexstr(a_response[29],2,TRUE));
						str_response:=concat(str_response,byte_to_hexstr(a_response[30],2,TRUE));
						str_response:=concat(str_response,byte_to_hexstr(a_response[31],2,TRUE));
						
					// "Digest username=\"admin\", realm=\"shellypro4pm-083af27cfbac\", nonce=\"63768368\", uri=\"/rpc/Switch.GetStatus?id=0\", algorithm=\"SHA-256\", qop=auth, nc=00000001, cnonce=\"oKOklSrS\", response=\"d1d59d1e015dee0a3acfc97b20a0fa0ff851b03d79ca00df59ce018a63041468\""
					
					str_authorization:=concat('Digest username="admin", realm="',sRealm);
					str_authorization:=concat(str_authorization,'", nonce="');
					str_authorization:=concat(str_authorization,snonce);
					str_authorization:=concat(str_authorization,'", algorithm="SHA-256", uri="/rpc/Switch.GetStatus?id=0", qop=auth, nc=00000001, cnonce="');
					str_authorization:=concat(str_authorization,scnonce);
					str_authorization:=concat(str_authorization,'", response="');
					str_authorization:=concat(str_authorization,str_response);
					str_authorization:=concat(str_authorization,'"');
					
					fbHeader.AddField('Authorization', str_authorization, FALSE);
					IF fbRequest2.SendRequest(sUri:= '/rpc/Switch.GetStatus?id=0', fbClient:= fbClient, eRequestType:= ETcIotHttpRequestType.HTTP_Get, 0, 0, fbHeader) THEN
						nState:= 2;
						bBusy:= TRUE;
						bError:= FALSE;
					END_IF
			END_IF
		END_IF
	END_IF


2:
	IF NOT fbRequest2.bBusy THEN
		bError:= TRUE;
		
		IF NOT fbRequest2.bError THEN				 
			bGetContentResult:= fbRequest2.GetContent(pContent:= ADR(sfincontent), nContentSize:= SIZEOF(sfincontent), bSetNullTermination:= TRUE);

			IF fbRequest2.nStatusCode >= 200 AND fbRequest2.nStatusCode < 300 THEN
				bGetJsonResult:= FALSE;
				jsonDoc:= fbRequest2.GetJsonDomContent(fbJson);
				IF jsonDoc <> 0 THEN
					bGetJsonResult:= TRUE;
					IF fbJson.HasMember(jsonDoc, 'output')  THEN
						jsonVal:= fbJson.FindMember(jsonDoc, 'output');
						nValidResCount:= nValidResCount+1;					
						IF fbJson.IsBool(jsonVal) AND (fbJson.GetBool(jsonVal)=TRUE OR fbJson.GetBool(jsonVal)=FALSE) THEN							
							bStateP1:= fbJson.GetBool(jsonVal);									
						END_IF
					END_IF
					IF fbJson.HasMember(jsonDoc, 'apower')  THEN
						jsonVal:= fbJson.FindMember(jsonDoc, 'apower');
						nValidResCount:= nValidResCount+1;
						IF fbJson.IsDouble(jsonVal) AND fbJson.GetDouble(jsonVal)> -3.402823E+38 AND fbJson.GetDouble(jsonVal)< 3.402823E+38 THEN							
							lrapowerP1:= fbJson.GetDouble(jsonVal);									
						END_IF
					END_IF
					IF fbJson.HasMember(jsonDoc, 'voltage')  THEN
						jsonVal:= fbJson.FindMember(jsonDoc, 'voltage');
						nValidResCount:= nValidResCount+1;					
						IF fbJson.IsDouble(jsonVal) AND fbJson.GetDouble(jsonVal)> -3.402823E+38 AND fbJson.GetDouble(jsonVal)< 3.402823E+38 THEN
							lrvoltageP1:= fbJson.GetDouble(jsonVal);									
						END_IF
					END_IF
					IF fbJson.HasMember(jsonDoc, 'temperature')  THEN
						jsonVal:= fbJson.FindMember(jsonDoc, 'temperature');
						 IF fbJson.HasMember(jsonVal, 'tC') AND fbJson.GetDouble(jsonVal)> -3.402823E+38 AND fbJson.GetDouble(jsonVal)< 3.402823E+38 THEN							
                            jsonVal:= fbJson.FindMember(jsonVal, 'tC');
							nValidResCount:= nValidResCount+1;					
							IF fbJson.IsDouble(jsonVal) AND fbJson.GetDouble(jsonVal)> -3.402823E+38 AND fbJson.GetDouble(jsonVal)< 3.402823E+38 THEN
								lrTemperatureP1:= fbJson.GetDouble(jsonVal);									
							END_IF
						END_IF
					END_IF
					IF fbJson.HasMember(jsonDoc, 'aenergy')  THEN
						jsonVal:= fbJson.FindMember(jsonDoc, 'aenergy');
                        IF fbJson.HasMember(jsonVal, 'total') AND fbJson.GetDouble(jsonVal)> -3.402823E+38 AND fbJson.GetDouble(jsonVal)< 3.402823E+38 THEN							
                            jsonVal:= fbJson.FindMember(jsonVal, 'total');
                            nValidResCount:= nValidResCount+1;
                            IF fbJson.IsDouble(jsonVal) AND fbJson.GetDouble(jsonVal)> -3.402823E+38 AND fbJson.GetDouble(jsonVal)< 3.402823E+38 THEN
                                lraenergyP1:= fbJson.GetDouble(jsonVal);
                            END_IF
						bError:= FALSE;
						END_IF
					END_IF	

				nResCount:= nResCount+1;			
				END_IF
			END_IF
		END_IF
		
	nState:= 0;
	bBusy:= FALSE;
		IF bError THEN
			nErrCount:= nErrCount+1;
		END_IF
	END_IF
	
END_CASE

END_FUNCTION_BLOCK

// ---- FBs/FB_Shelly_Pro1PM_Helper_2.TcPOU
FUNCTION_BLOCK FB_Shelly_Pro1PM_Helper_2
VAR_INPUT
	bSend			: BOOL;
	bSetOnP1		: BOOL;
	bSetOffP1		: BOOL;
END_VAR

VAR_IN_OUT
	fbClient		: FB_IotHttpClient;
END_VAR

VAR_OUTPUT
	bBusy			: BOOL;
	bError			: BOOL;
	bStateP1		: BOOL;
	lrapowerP1		: LREAL;
	lrvoltageP1		: LREAL;
	lraenergyP1		: LREAL;
	lrTemperatureP1	: LREAL;
END_VAR

VAR
	fbRequestSwitch0	: FB_IotHttpRequest;
	RisingEdge			: R_TRIG;
	RisingEdgeSetOnP1	: R_TRIG;
	RisingEdgeSetOffP1	: R_TRIG;
	fbJson				: FB_JsonDomParser;
	nState				: UDINT;
	timTimeout			: TON;
	tTimeOut			: TIME := T#30S;
	timTimeoutSwitch	: TON;
	tTimeOutSwitch		: TIME := T#5S;
	bGetContentResult	: BOOL;
	sContentS0			: STRING(511);
	
	bGetJsonResult		: BOOL;
	jsonDoc				: SJsonValue;
	jsonVal				: SJsonValue;
	
	nReqCount			: UDINT;	
	nResCount			: UDINT;
	nValidResCount		: UDINT;
	nErrCount			: UDINT;
	
	fbRequest2         : FB_IotHttpRequest;
	fbRequest3         : FB_IotHttpRequest;
	fbHeader            : FB_IotHttpHeaderFieldMap;
	
	sRealm	:	STRING(511);
	sPassword :	STRING(511) := ':sh3lly4ankerio2$$';
	snonce	:	STRING(511);
	scnonce	:	STRING(511);
	shash	: STRING(511);
	bhash	: BOOL;
	
	aData	: STRING(511);
	a_ha1	: ARRAY[0..31] OF BYTE;
	str_ha1 : STRING(511);
	str_Toha1   : STRING(511);
	udint_length_string : UDINT;
	
	a_ha2	: ARRAY[0..31] OF BYTE;
	str_ha2 : STRING(511);
	str_Toha2   : STRING(511);
	
	a_response	: ARRAY[0..31] OF BYTE;
	str_response : STRING(511);
	str_Toresponse   : STRING(511);

	str_authorization	: STRING(2048);
	
	sfincontent	: STRING(511);
	int_CountOffWrite: INT;
	int_CountOnWrite: INT;
END_VAR

//Timer for Timeout
timTimeout(IN:= nState = 1 AND bBusy, PT:= tTimeOut, Q=> , ET=> );
	IF timTimeout.Q THEN 
		nState := 0;
		bBusy := FALSE;
	END_IF
	
timTimeoutSwitch(IN:= bSetOnP1 OR bSetOffP1, PT:= tTimeOut, Q=> , ET=> );
	IF timTimeoutSwitch.Q THEN 
		bSetOnP1 := FALSE;
		bSetOffP1 := FALSE;
	END_IF

RisingEdge(CLK:= bSend );
RisingEdgeSetOnP1(CLK:= bSetOnP1 );
RisingEdgeSetOffP1(CLK:= bSetOffP1 );

CASE nState OF
	0:	
		IF RisingEdge.Q THEN 
			IF
				fbRequestSwitch0.SendRequest(sUri:='/rpc/Switch.GetStatus?id=0', fbClient:=fbClient, eRequestType:=ETcIotHttpRequestType.HTTP_Get, 0, 0, 0) THEN
				nState:= 1;
				nReqCount:= nReqCount+1;
				bBusy:= TRUE;
				bError:= FALSE;
			END_IF					
		END_IF
	1:
		IF NOT fbRequestSwitch0.bBusy THEN
			bError:= TRUE;
			IF NOT fbRequestSwitch0.bError THEN
				bGetContentResult:= fbRequestSwitch0.GetHeaderField(pValue:= ADR(sContentS0), 
														 nValueSize:= SIZEOF(sContentS0), sField := 'WWW-Authenticate');
				IF fbRequestSwitch0.nStatusCode = 401 THEN
					bGetJsonResult:= FALSE;
						sRealm := sContentS0;
						sRealm := DELETE(sRealm, FIND(sRealm, 'realm') + 7, 0);
						sRealm := DELETE(sRealm, LEN(sRealm), FIND(sRealm, '"'));
						
						snonce := sContentS0;
						snonce := DELETE(snonce, FIND(snonce, 'nonce') + 7, 0);
						snonce := DELETE(snonce, LEN(snonce), FIND(snonce, '"'));
						
						scnonce := 'YmawvYzT';
					
						aData := sRealm;
						
						str_Toha1:=concat('admin:', sRealm);
						str_Toha1:=concat(str_Toha1, sPassword);
		 
						udint_length_string:= len2(ADR(str_Toha1));
						F_GenerateHashValue(E_HashMode.HASH_SHA256,ADR(str_Toha1),udint_length_string,ADR(a_ha1),32);
						
							str_ha1:=concat(byte_to_hexstr(a_ha1[0],2,TRUE),byte_to_hexstr(a_ha1[1],2,TRUE));
							str_ha1:=concat(str_ha1,byte_to_hexstr(a_ha1[2],2,TRUE));
							str_ha1:=concat(str_ha1,byte_to_hexstr(a_ha1[3],2,TRUE));
							str_ha1:=concat(str_ha1,byte_to_hexstr(a_ha1[4],2,TRUE));
							str_ha1:=concat(str_ha1,byte_to_hexstr(a_ha1[5],2,TRUE));
							str_ha1:=concat(str_ha1,byte_to_hexstr(a_ha1[6],2,TRUE));
							str_ha1:=concat(str_ha1,byte_to_hexstr(a_ha1[7],2,TRUE));
							str_ha1:=concat(str_ha1,byte_to_hexstr(a_ha1[8],2,TRUE));
							str_ha1:=concat(str_ha1,byte_to_hexstr(a_ha1[9],2,TRUE));
							str_ha1:=concat(str_ha1,byte_to_hexstr(a_ha1[10],2,TRUE));
							str_ha1:=concat(str_ha1,byte_to_hexstr(a_ha1[11],2,TRUE));
							str_ha1:=concat(str_ha1,byte_to_hexstr(a_ha1[12],2,TRUE));
							str_ha1:=concat(str_ha1,byte_to_hexstr(a_ha1[13],2,TRUE));
							str_ha1:=concat(str_ha1,byte_to_hexstr(a_ha1[14],2,TRUE));
							str_ha1:=concat(str_ha1,byte_to_hexstr(a_ha1[15],2,TRUE));
							str_ha1:=concat(str_ha1,byte_to_hexstr(a_ha1[16],2,TRUE));
							str_ha1:=concat(str_ha1,byte_to_hexstr(a_ha1[17],2,TRUE));
							str_ha1:=concat(str_ha1,byte_to_hexstr(a_ha1[18],2,TRUE));
							str_ha1:=concat(str_ha1,byte_to_hexstr(a_ha1[19],2,TRUE));
							str_ha1:=concat(str_ha1,byte_to_hexstr(a_ha1[20],2,TRUE));
							str_ha1:=concat(str_ha1,byte_to_hexstr(a_ha1[21],2,TRUE));
							str_ha1:=concat(str_ha1,byte_to_hexstr(a_ha1[22],2,TRUE));
							str_ha1:=concat(str_ha1,byte_to_hexstr(a_ha1[23],2,TRUE));
							str_ha1:=concat(str_ha1,byte_to_hexstr(a_ha1[24],2,TRUE));
							str_ha1:=concat(str_ha1,byte_to_hexstr(a_ha1[25],2,TRUE));
							str_ha1:=concat(str_ha1,byte_to_hexstr(a_ha1[26],2,TRUE));
							str_ha1:=concat(str_ha1,byte_to_hexstr(a_ha1[27],2,TRUE));
							str_ha1:=concat(str_ha1,byte_to_hexstr(a_ha1[28],2,TRUE));
							str_ha1:=concat(str_ha1,byte_to_hexstr(a_ha1[29],2,TRUE));
							str_ha1:=concat(str_ha1,byte_to_hexstr(a_ha1[30],2,TRUE));
							str_ha1:=concat(str_ha1,byte_to_hexstr(a_ha1[31],2,TRUE));
						
						str_Toha2:='GET:/rpc/Switch.GetStatus?id=0';
		 
						udint_length_string:= len2(ADR(str_Toha2));
						F_GenerateHashValue(E_HashMode.HASH_SHA256,ADR(str_Toha2),udint_length_string,ADR(a_ha2),32);
						
							str_ha2:=concat(byte_to_hexstr(a_ha2[0],2,TRUE),byte_to_hexstr(a_ha2[1],2,TRUE));
							str_ha2:=concat(str_ha2,byte_to_hexstr(a_ha2[2],2,TRUE));
							str_ha2:=concat(str_ha2,byte_to_hexstr(a_ha2[3],2,TRUE));
							str_ha2:=concat(str_ha2,byte_to_hexstr(a_ha2[4],2,TRUE));
							str_ha2:=concat(str_ha2,byte_to_hexstr(a_ha2[5],2,TRUE));
							str_ha2:=concat(str_ha2,byte_to_hexstr(a_ha2[6],2,TRUE));
							str_ha2:=concat(str_ha2,byte_to_hexstr(a_ha2[7],2,TRUE));
							str_ha2:=concat(str_ha2,byte_to_hexstr(a_ha2[8],2,TRUE));
							str_ha2:=concat(str_ha2,byte_to_hexstr(a_ha2[9],2,TRUE));
							str_ha2:=concat(str_ha2,byte_to_hexstr(a_ha2[10],2,TRUE));
							str_ha2:=concat(str_ha2,byte_to_hexstr(a_ha2[11],2,TRUE));
							str_ha2:=concat(str_ha2,byte_to_hexstr(a_ha2[12],2,TRUE));
							str_ha2:=concat(str_ha2,byte_to_hexstr(a_ha2[13],2,TRUE));
							str_ha2:=concat(str_ha2,byte_to_hexstr(a_ha2[14],2,TRUE));
							str_ha2:=concat(str_ha2,byte_to_hexstr(a_ha2[15],2,TRUE));
							str_ha2:=concat(str_ha2,byte_to_hexstr(a_ha2[16],2,TRUE));
							str_ha2:=concat(str_ha2,byte_to_hexstr(a_ha2[17],2,TRUE));
							str_ha2:=concat(str_ha2,byte_to_hexstr(a_ha2[18],2,TRUE));
							str_ha2:=concat(str_ha2,byte_to_hexstr(a_ha2[19],2,TRUE));
							str_ha2:=concat(str_ha2,byte_to_hexstr(a_ha2[20],2,TRUE));
							str_ha2:=concat(str_ha2,byte_to_hexstr(a_ha2[21],2,TRUE));
							str_ha2:=concat(str_ha2,byte_to_hexstr(a_ha2[22],2,TRUE));
							str_ha2:=concat(str_ha2,byte_to_hexstr(a_ha2[23],2,TRUE));
							str_ha2:=concat(str_ha2,byte_to_hexstr(a_ha2[24],2,TRUE));
							str_ha2:=concat(str_ha2,byte_to_hexstr(a_ha2[25],2,TRUE));
							str_ha2:=concat(str_ha2,byte_to_hexstr(a_ha2[26],2,TRUE));
							str_ha2:=concat(str_ha2,byte_to_hexstr(a_ha2[27],2,TRUE));
							str_ha2:=concat(str_ha2,byte_to_hexstr(a_ha2[28],2,TRUE));
							str_ha2:=concat(str_ha2,byte_to_hexstr(a_ha2[29],2,TRUE));
							str_ha2:=concat(str_ha2,byte_to_hexstr(a_ha2[30],2,TRUE));
							str_ha2:=concat(str_ha2,byte_to_hexstr(a_ha2[31],2,TRUE));
							
						// <ha1> + ":" + <nonce> + ":" + <nc> + ":" + <cnonce> + ":" + "auth" + ":" + <ha2>
						
						str_Toresponse:=concat(str_ha1,':');
						str_Toresponse:=concat(str_Toresponse,snonce);
						str_Toresponse:=concat(str_Toresponse,':00000001:');
						str_Toresponse:=concat(str_Toresponse,scnonce);
						str_Toresponse:=concat(str_Toresponse,':');
						str_Toresponse:=concat(str_Toresponse,'auth:');
						str_Toresponse:=concat(str_Toresponse,str_ha2);
						
						udint_length_string:= len2(ADR(str_Toresponse));
						F_GenerateHashValue(E_HashMode.HASH_SHA256,ADR(str_Toresponse),udint_length_string,ADR(a_response),32);
						
							str_response:=concat(byte_to_hexstr(a_response[0],2,TRUE),byte_to_hexstr(a_response[1],2,TRUE));
							str_response:=concat(str_response,byte_to_hexstr(a_response[2],2,TRUE));
							str_response:=concat(str_response,byte_to_hexstr(a_response[3],2,TRUE));
							str_response:=concat(str_response,byte_to_hexstr(a_response[4],2,TRUE));
							str_response:=concat(str_response,byte_to_hexstr(a_response[5],2,TRUE));
							str_response:=concat(str_response,byte_to_hexstr(a_response[6],2,TRUE));
							str_response:=concat(str_response,byte_to_hexstr(a_response[7],2,TRUE));
							str_response:=concat(str_response,byte_to_hexstr(a_response[8],2,TRUE));
							str_response:=concat(str_response,byte_to_hexstr(a_response[9],2,TRUE));
							str_response:=concat(str_response,byte_to_hexstr(a_response[10],2,TRUE));
							str_response:=concat(str_response,byte_to_hexstr(a_response[11],2,TRUE));
							str_response:=concat(str_response,byte_to_hexstr(a_response[12],2,TRUE));
							str_response:=concat(str_response,byte_to_hexstr(a_response[13],2,TRUE));
							str_response:=concat(str_response,byte_to_hexstr(a_response[14],2,TRUE));
							str_response:=concat(str_response,byte_to_hexstr(a_response[15],2,TRUE));
							str_response:=concat(str_response,byte_to_hexstr(a_response[16],2,TRUE));
							str_response:=concat(str_response,byte_to_hexstr(a_response[17],2,TRUE));
							str_response:=concat(str_response,byte_to_hexstr(a_response[18],2,TRUE));
							str_response:=concat(str_response,byte_to_hexstr(a_response[19],2,TRUE));
							str_response:=concat(str_response,byte_to_hexstr(a_response[20],2,TRUE));
							str_response:=concat(str_response,byte_to_hexstr(a_response[21],2,TRUE));
							str_response:=concat(str_response,byte_to_hexstr(a_response[22],2,TRUE));
							str_response:=concat(str_response,byte_to_hexstr(a_response[23],2,TRUE));
							str_response:=concat(str_response,byte_to_hexstr(a_response[24],2,TRUE));
							str_response:=concat(str_response,byte_to_hexstr(a_response[25],2,TRUE));
							str_response:=concat(str_response,byte_to_hexstr(a_response[26],2,TRUE));
							str_response:=concat(str_response,byte_to_hexstr(a_response[27],2,TRUE));
							str_response:=concat(str_response,byte_to_hexstr(a_response[28],2,TRUE));
							str_response:=concat(str_response,byte_to_hexstr(a_response[29],2,TRUE));
							str_response:=concat(str_response,byte_to_hexstr(a_response[30],2,TRUE));
							str_response:=concat(str_response,byte_to_hexstr(a_response[31],2,TRUE));
							
						// "Digest username=\"admin\", realm=\"shellypro4pm-083af27cfbac\", nonce=\"63768368\", uri=\"/rpc/Switch.GetStatus?id=0\", algorithm=\"SHA-256\", qop=auth, nc=00000001, cnonce=\"oKOklSrS\", response=\"d1d59d1e015dee0a3acfc97b20a0fa0ff851b03d79ca00df59ce018a63041468\""
						
						str_authorization:=concat('Digest username="admin", realm="',sRealm);
						str_authorization:=concat(str_authorization,'", nonce="');
						str_authorization:=concat(str_authorization,snonce);
						str_authorization:=concat(str_authorization,'", algorithm="SHA-256", uri="/rpc/Switch.GetStatus?id=0", qop=auth, nc=00000001, cnonce="');
						str_authorization:=concat(str_authorization,scnonce);
						str_authorization:=concat(str_authorization,'", response="');
						str_authorization:=concat(str_authorization,str_response);
						str_authorization:=concat(str_authorization,'"');
						
						fbHeader.AddField('Authorization', str_authorization, FALSE);
						IF fbRequest2.SendRequest(sUri:= '/rpc/Switch.GetStatus?id=0', fbClient:= fbClient, eRequestType:= ETcIotHttpRequestType.HTTP_Get, 0, 0, fbHeader) THEN
							nState:= 2;
							bBusy:= TRUE;
							bError:= FALSE;
						END_IF
				END_IF
			END_IF
		END_IF
	
	
	2:
		IF NOT fbRequest2.bBusy THEN
			bError:= TRUE;
			
			IF NOT fbRequest2.bError THEN				 
				bGetContentResult:= fbRequest2.GetContent(pContent:= ADR(sfincontent), nContentSize:= SIZEOF(sfincontent), bSetNullTermination:= TRUE);
	
				IF fbRequest2.nStatusCode >= 200 AND fbRequest2.nStatusCode < 300 THEN
					bGetJsonResult:= FALSE;
					jsonDoc:= fbRequest2.GetJsonDomContent(fbJson);
					IF jsonDoc <> 0 THEN
						bGetJsonResult:= TRUE;
						IF fbJson.HasMember(jsonDoc, 'output')  THEN
							jsonVal:= fbJson.FindMember(jsonDoc, 'output');
							nValidResCount:= nValidResCount+1;					
							IF fbJson.IsBool(jsonVal) AND (fbJson.GetBool(jsonVal)=TRUE OR fbJson.GetBool(jsonVal)=FALSE) THEN							
								bStateP1:= fbJson.GetBool(jsonVal);									
							END_IF
						END_IF
						IF fbJson.HasMember(jsonDoc, 'apower')  THEN
							jsonVal:= fbJson.FindMember(jsonDoc, 'apower');
							nValidResCount:= nValidResCount+1;
							IF fbJson.IsDouble(jsonVal) AND fbJson.GetDouble(jsonVal)> -3.402823E+38 AND fbJson.GetDouble(jsonVal)< 3.402823E+38 THEN							
								lrapowerP1:= fbJson.GetDouble(jsonVal);									
							END_IF
						END_IF
						IF fbJson.HasMember(jsonDoc, 'voltage')  THEN
							jsonVal:= fbJson.FindMember(jsonDoc, 'voltage');
							nValidResCount:= nValidResCount+1;					
							IF fbJson.IsDouble(jsonVal) AND fbJson.GetDouble(jsonVal)> -3.402823E+38 AND fbJson.GetDouble(jsonVal)< 3.402823E+38 THEN
								lrvoltageP1:= fbJson.GetDouble(jsonVal);									
							END_IF
						END_IF
						IF fbJson.HasMember(jsonDoc, 'temperature')  THEN
							jsonVal:= fbJson.FindMember(jsonDoc, 'temperature');
							 IF fbJson.HasMember(jsonVal, 'tC') AND fbJson.GetDouble(jsonVal)> -3.402823E+38 AND fbJson.GetDouble(jsonVal)< 3.402823E+38 THEN							
								jsonVal:= fbJson.FindMember(jsonVal, 'tC');
								nValidResCount:= nValidResCount+1;					
								IF fbJson.IsDouble(jsonVal) AND fbJson.GetDouble(jsonVal)> -3.402823E+38 AND fbJson.GetDouble(jsonVal)< 3.402823E+38 THEN
									lrTemperatureP1:= fbJson.GetDouble(jsonVal);									
								END_IF
							END_IF
						END_IF
						IF fbJson.HasMember(jsonDoc, 'aenergy')  THEN
							jsonVal:= fbJson.FindMember(jsonDoc, 'aenergy');
							IF fbJson.HasMember(jsonVal, 'total') AND fbJson.GetDouble(jsonVal)> -3.402823E+38 AND fbJson.GetDouble(jsonVal)< 3.402823E+38 THEN							
								jsonVal:= fbJson.FindMember(jsonVal, 'total');
								nValidResCount:= nValidResCount+1;
								IF fbJson.IsDouble(jsonVal) AND fbJson.GetDouble(jsonVal)> -3.402823E+38 AND fbJson.GetDouble(jsonVal)< 3.402823E+38 THEN
									lraenergyP1:= fbJson.GetDouble(jsonVal);
								END_IF
							bError:= FALSE;
							END_IF
						END_IF	
					nResCount:= nResCount+1;			
					END_IF
				END_IF
			END_IF
			
		nState:= 3;
		bBusy:= FALSE;
			IF bError THEN
				nErrCount:= nErrCount+1;
			END_IF
		END_IF
	
	
	3:
		IF fbRequest3.SendRequest(sUri:= '/rpc/Switch.GetStatus?id=0', fbClient:= fbClient, eRequestType:= ETcIotHttpRequestType.HTTP_Get, 0, 0, fbHeader) THEN
			nState:= 4;
		END_IF

	4:	
		IF bSetOnP1 AND NOT bStateP1 THEN 
			IF
				fbRequest3.SendRequest(sUri:='/rpc/Switch.Set?id=0&on=true', fbClient:=fbClient, eRequestType:=ETcIotHttpRequestType.HTTP_Get, 0, 0, fbHeader) THEN				
				bSetOnP1 := FALSE;
				int_CountOnWrite := int_CountOnWrite +1;
				nState:= 5;
				bBusy:= TRUE;
				bError:= FALSE;
			END_IF					
		ELSIF bSetOffP1 AND bStateP1 THEN 
			IF	
				fbRequest3.SendRequest(sUri:='/rpc/Switch.Set?id=0&on=false', fbClient:=fbClient, eRequestType:=ETcIotHttpRequestType.HTTP_Get, 0, 0, fbHeader) THEN				
				bSetOffP1 := FALSE;
				int_CountOffWrite := int_CountOffWrite +1;
				nState:= 5;
				bBusy:= TRUE;
				bError:= FALSE;
			END_IF	
		ELSE
			nState:= 5;
		END_IF
	5:
		bBusy:= FALSE;
		nState:= 0;

	
END_CASE

END_FUNCTION_BLOCK

// ---- FBs/FB_Shelly_Pro1PM_Helper_3.TcPOU
FUNCTION_BLOCK FB_Shelly_Pro1PM_Helper_3
VAR_INPUT
	bSend			: BOOL;
	bSetOnP1		: BOOL;
	bSetOffP1		: BOOL;
END_VAR

VAR_IN_OUT
	fbClient		: FB_IotHttpClient;
END_VAR

VAR_OUTPUT
	bBusy			: BOOL;
	bError			: BOOL;
	bStateP1		: BOOL;
	lrapowerP1		: LREAL;
	lrvoltageP1		: LREAL;
	lraenergyP1		: LREAL;
	lrTemperatureP1	: LREAL;
END_VAR

VAR
	fbRequestSwitch0	: FB_IotHttpRequest;
	fbRequestSwitch1	: FB_IotHttpRequest;
	RisingEdge			: R_TRIG;
	RisingEdgeSetOnP1	: R_TRIG;
	RisingEdgeSetOffP1	: R_TRIG;
	fbJson				: FB_JsonDomParser;
	nState				: UDINT;
	timTimeout			: TON;
	tTimeOut			: TIME := T#30S;
	timTimeoutSwitch	: TON;
	tTimeOutSwitch		: TIME := T#5S;
	bGetContentResult	: BOOL;
	sContentS0			: STRING(511);
	
	bGetJsonResult		: BOOL;
	jsonDoc				: SJsonValue;
	jsonVal				: SJsonValue;
	
	nReqCount			: UDINT;	
	nResCount			: UDINT;
	nValidResCount		: UDINT;
	nErrCount			: UDINT;
	
	fbRequest2         : FB_IotHttpRequest;
	fbRequest3         : FB_IotHttpRequest;
	fbHeader            : FB_IotHttpHeaderFieldMap;
	fbHeader2            : FB_IotHttpHeaderFieldMap;
	
	sRealm	:	STRING(511);
	sPassword :	STRING(511) := ':sh3lly4ankerio2$$';
	snonce	:	STRING(511);
	scnonce	:	STRING(511);
	shash	: STRING(511);
	bhash	: BOOL;
	
	aData	: STRING(511);
	a_ha1	: ARRAY[0..31] OF BYTE;
	str_ha1 : STRING(511);
	str_Toha1   : STRING(511);
	udint_length_string : UDINT;
	
	a_ha2	: ARRAY[0..31] OF BYTE;
	str_ha2 : STRING(511);
	str_Toha2   : STRING(511);
	
	a_response	: ARRAY[0..31] OF BYTE;
	str_response : STRING(511);
	str_Toresponse   : STRING(511);

	str_authorization	: STRING(2048);
	
	sfincontent	: STRING(511);
	int_CountOffWrite: INT;
	int_CountOnWrite: INT;
END_VAR

//Timer for Timeout
timTimeout(IN:= nState = 1 AND bBusy, PT:= tTimeOut, Q=> , ET=> );
	IF timTimeout.Q THEN 
		nState := 0;
		bBusy := FALSE;
	END_IF
	
timTimeoutSwitch(IN:= bSetOnP1 OR bSetOffP1, PT:= tTimeOut, Q=> , ET=> );
	IF timTimeoutSwitch.Q THEN 
		bSetOnP1 := FALSE;
		bSetOffP1 := FALSE;
	END_IF

RisingEdge(CLK:= bSend );
RisingEdgeSetOnP1(CLK:= bSetOnP1 );
RisingEdgeSetOffP1(CLK:= bSetOffP1 );

CASE nState OF
	0:	
		IF RisingEdge.Q THEN 
			IF
				fbRequestSwitch0.SendRequest(sUri:='/rpc/Switch.GetStatus?id=0', fbClient:=fbClient, eRequestType:=ETcIotHttpRequestType.HTTP_Get, 0, 0, 0) THEN
				nState:= 1;
				nReqCount:= nReqCount+1;
				bBusy:= TRUE;
				bError:= FALSE;
			END_IF
		END_IF
	1:
		IF NOT fbRequestSwitch0.bBusy THEN
			bError:= TRUE;
			IF NOT fbRequestSwitch0.bError THEN
				bGetContentResult:= fbRequestSwitch0.GetHeaderField(pValue:= ADR(sContentS0), 
														 nValueSize:= SIZEOF(sContentS0), sField := 'WWW-Authenticate');
				IF fbRequestSwitch0.nStatusCode = 401 THEN
					bGetJsonResult:= FALSE;
						sRealm := sContentS0;
						sRealm := DELETE(sRealm, FIND(sRealm, 'realm') + 7, 0);
						sRealm := DELETE(sRealm, LEN(sRealm), FIND(sRealm, '"'));
						
						snonce := sContentS0;
						snonce := DELETE(snonce, FIND(snonce, 'nonce') + 7, 0);
						snonce := DELETE(snonce, LEN(snonce), FIND(snonce, '"'));
						
						scnonce := 'YmawvYzT';
					
						aData := sRealm;
						
						str_Toha1:=concat('admin:', sRealm);
						str_Toha1:=concat(str_Toha1, sPassword);
		 
						udint_length_string:= len2(ADR(str_Toha1));
						F_GenerateHashValue(E_HashMode.HASH_SHA256,ADR(str_Toha1),udint_length_string,ADR(a_ha1),32);
						
							str_ha1:=concat(byte_to_hexstr(a_ha1[0],2,TRUE),byte_to_hexstr(a_ha1[1],2,TRUE));
							str_ha1:=concat(str_ha1,byte_to_hexstr(a_ha1[2],2,TRUE));
							str_ha1:=concat(str_ha1,byte_to_hexstr(a_ha1[3],2,TRUE));
							str_ha1:=concat(str_ha1,byte_to_hexstr(a_ha1[4],2,TRUE));
							str_ha1:=concat(str_ha1,byte_to_hexstr(a_ha1[5],2,TRUE));
							str_ha1:=concat(str_ha1,byte_to_hexstr(a_ha1[6],2,TRUE));
							str_ha1:=concat(str_ha1,byte_to_hexstr(a_ha1[7],2,TRUE));
							str_ha1:=concat(str_ha1,byte_to_hexstr(a_ha1[8],2,TRUE));
							str_ha1:=concat(str_ha1,byte_to_hexstr(a_ha1[9],2,TRUE));
							str_ha1:=concat(str_ha1,byte_to_hexstr(a_ha1[10],2,TRUE));
							str_ha1:=concat(str_ha1,byte_to_hexstr(a_ha1[11],2,TRUE));
							str_ha1:=concat(str_ha1,byte_to_hexstr(a_ha1[12],2,TRUE));
							str_ha1:=concat(str_ha1,byte_to_hexstr(a_ha1[13],2,TRUE));
							str_ha1:=concat(str_ha1,byte_to_hexstr(a_ha1[14],2,TRUE));
							str_ha1:=concat(str_ha1,byte_to_hexstr(a_ha1[15],2,TRUE));
							str_ha1:=concat(str_ha1,byte_to_hexstr(a_ha1[16],2,TRUE));
							str_ha1:=concat(str_ha1,byte_to_hexstr(a_ha1[17],2,TRUE));
							str_ha1:=concat(str_ha1,byte_to_hexstr(a_ha1[18],2,TRUE));
							str_ha1:=concat(str_ha1,byte_to_hexstr(a_ha1[19],2,TRUE));
							str_ha1:=concat(str_ha1,byte_to_hexstr(a_ha1[20],2,TRUE));
							str_ha1:=concat(str_ha1,byte_to_hexstr(a_ha1[21],2,TRUE));
							str_ha1:=concat(str_ha1,byte_to_hexstr(a_ha1[22],2,TRUE));
							str_ha1:=concat(str_ha1,byte_to_hexstr(a_ha1[23],2,TRUE));
							str_ha1:=concat(str_ha1,byte_to_hexstr(a_ha1[24],2,TRUE));
							str_ha1:=concat(str_ha1,byte_to_hexstr(a_ha1[25],2,TRUE));
							str_ha1:=concat(str_ha1,byte_to_hexstr(a_ha1[26],2,TRUE));
							str_ha1:=concat(str_ha1,byte_to_hexstr(a_ha1[27],2,TRUE));
							str_ha1:=concat(str_ha1,byte_to_hexstr(a_ha1[28],2,TRUE));
							str_ha1:=concat(str_ha1,byte_to_hexstr(a_ha1[29],2,TRUE));
							str_ha1:=concat(str_ha1,byte_to_hexstr(a_ha1[30],2,TRUE));
							str_ha1:=concat(str_ha1,byte_to_hexstr(a_ha1[31],2,TRUE));
						
						str_Toha2:='GET:/rpc/Switch.GetStatus?id=0';
		 
						udint_length_string:= len2(ADR(str_Toha2));
						F_GenerateHashValue(E_HashMode.HASH_SHA256,ADR(str_Toha2),udint_length_string,ADR(a_ha2),32);
						
							str_ha2:=concat(byte_to_hexstr(a_ha2[0],2,TRUE),byte_to_hexstr(a_ha2[1],2,TRUE));
							str_ha2:=concat(str_ha2,byte_to_hexstr(a_ha2[2],2,TRUE));
							str_ha2:=concat(str_ha2,byte_to_hexstr(a_ha2[3],2,TRUE));
							str_ha2:=concat(str_ha2,byte_to_hexstr(a_ha2[4],2,TRUE));
							str_ha2:=concat(str_ha2,byte_to_hexstr(a_ha2[5],2,TRUE));
							str_ha2:=concat(str_ha2,byte_to_hexstr(a_ha2[6],2,TRUE));
							str_ha2:=concat(str_ha2,byte_to_hexstr(a_ha2[7],2,TRUE));
							str_ha2:=concat(str_ha2,byte_to_hexstr(a_ha2[8],2,TRUE));
							str_ha2:=concat(str_ha2,byte_to_hexstr(a_ha2[9],2,TRUE));
							str_ha2:=concat(str_ha2,byte_to_hexstr(a_ha2[10],2,TRUE));
							str_ha2:=concat(str_ha2,byte_to_hexstr(a_ha2[11],2,TRUE));
							str_ha2:=concat(str_ha2,byte_to_hexstr(a_ha2[12],2,TRUE));
							str_ha2:=concat(str_ha2,byte_to_hexstr(a_ha2[13],2,TRUE));
							str_ha2:=concat(str_ha2,byte_to_hexstr(a_ha2[14],2,TRUE));
							str_ha2:=concat(str_ha2,byte_to_hexstr(a_ha2[15],2,TRUE));
							str_ha2:=concat(str_ha2,byte_to_hexstr(a_ha2[16],2,TRUE));
							str_ha2:=concat(str_ha2,byte_to_hexstr(a_ha2[17],2,TRUE));
							str_ha2:=concat(str_ha2,byte_to_hexstr(a_ha2[18],2,TRUE));
							str_ha2:=concat(str_ha2,byte_to_hexstr(a_ha2[19],2,TRUE));
							str_ha2:=concat(str_ha2,byte_to_hexstr(a_ha2[20],2,TRUE));
							str_ha2:=concat(str_ha2,byte_to_hexstr(a_ha2[21],2,TRUE));
							str_ha2:=concat(str_ha2,byte_to_hexstr(a_ha2[22],2,TRUE));
							str_ha2:=concat(str_ha2,byte_to_hexstr(a_ha2[23],2,TRUE));
							str_ha2:=concat(str_ha2,byte_to_hexstr(a_ha2[24],2,TRUE));
							str_ha2:=concat(str_ha2,byte_to_hexstr(a_ha2[25],2,TRUE));
							str_ha2:=concat(str_ha2,byte_to_hexstr(a_ha2[26],2,TRUE));
							str_ha2:=concat(str_ha2,byte_to_hexstr(a_ha2[27],2,TRUE));
							str_ha2:=concat(str_ha2,byte_to_hexstr(a_ha2[28],2,TRUE));
							str_ha2:=concat(str_ha2,byte_to_hexstr(a_ha2[29],2,TRUE));
							str_ha2:=concat(str_ha2,byte_to_hexstr(a_ha2[30],2,TRUE));
							str_ha2:=concat(str_ha2,byte_to_hexstr(a_ha2[31],2,TRUE));
							
						// <ha1> + ":" + <nonce> + ":" + <nc> + ":" + <cnonce> + ":" + "auth" + ":" + <ha2>
						
						str_Toresponse:=concat(str_ha1,':');
						str_Toresponse:=concat(str_Toresponse,snonce);
						str_Toresponse:=concat(str_Toresponse,':00000001:');
						str_Toresponse:=concat(str_Toresponse,scnonce);
						str_Toresponse:=concat(str_Toresponse,':');
						str_Toresponse:=concat(str_Toresponse,'auth:');
						str_Toresponse:=concat(str_Toresponse,str_ha2);
						
						udint_length_string:= len2(ADR(str_Toresponse));
						F_GenerateHashValue(E_HashMode.HASH_SHA256,ADR(str_Toresponse),udint_length_string,ADR(a_response),32);
						
							str_response:=concat(byte_to_hexstr(a_response[0],2,TRUE),byte_to_hexstr(a_response[1],2,TRUE));
							str_response:=concat(str_response,byte_to_hexstr(a_response[2],2,TRUE));
							str_response:=concat(str_response,byte_to_hexstr(a_response[3],2,TRUE));
							str_response:=concat(str_response,byte_to_hexstr(a_response[4],2,TRUE));
							str_response:=concat(str_response,byte_to_hexstr(a_response[5],2,TRUE));
							str_response:=concat(str_response,byte_to_hexstr(a_response[6],2,TRUE));
							str_response:=concat(str_response,byte_to_hexstr(a_response[7],2,TRUE));
							str_response:=concat(str_response,byte_to_hexstr(a_response[8],2,TRUE));
							str_response:=concat(str_response,byte_to_hexstr(a_response[9],2,TRUE));
							str_response:=concat(str_response,byte_to_hexstr(a_response[10],2,TRUE));
							str_response:=concat(str_response,byte_to_hexstr(a_response[11],2,TRUE));
							str_response:=concat(str_response,byte_to_hexstr(a_response[12],2,TRUE));
							str_response:=concat(str_response,byte_to_hexstr(a_response[13],2,TRUE));
							str_response:=concat(str_response,byte_to_hexstr(a_response[14],2,TRUE));
							str_response:=concat(str_response,byte_to_hexstr(a_response[15],2,TRUE));
							str_response:=concat(str_response,byte_to_hexstr(a_response[16],2,TRUE));
							str_response:=concat(str_response,byte_to_hexstr(a_response[17],2,TRUE));
							str_response:=concat(str_response,byte_to_hexstr(a_response[18],2,TRUE));
							str_response:=concat(str_response,byte_to_hexstr(a_response[19],2,TRUE));
							str_response:=concat(str_response,byte_to_hexstr(a_response[20],2,TRUE));
							str_response:=concat(str_response,byte_to_hexstr(a_response[21],2,TRUE));
							str_response:=concat(str_response,byte_to_hexstr(a_response[22],2,TRUE));
							str_response:=concat(str_response,byte_to_hexstr(a_response[23],2,TRUE));
							str_response:=concat(str_response,byte_to_hexstr(a_response[24],2,TRUE));
							str_response:=concat(str_response,byte_to_hexstr(a_response[25],2,TRUE));
							str_response:=concat(str_response,byte_to_hexstr(a_response[26],2,TRUE));
							str_response:=concat(str_response,byte_to_hexstr(a_response[27],2,TRUE));
							str_response:=concat(str_response,byte_to_hexstr(a_response[28],2,TRUE));
							str_response:=concat(str_response,byte_to_hexstr(a_response[29],2,TRUE));
							str_response:=concat(str_response,byte_to_hexstr(a_response[30],2,TRUE));
							str_response:=concat(str_response,byte_to_hexstr(a_response[31],2,TRUE));
							
						// "Digest username=\"admin\", realm=\"shellypro4pm-083af27cfbac\", nonce=\"63768368\", uri=\"/rpc/Switch.GetStatus?id=0\", algorithm=\"SHA-256\", qop=auth, nc=00000001, cnonce=\"oKOklSrS\", response=\"d1d59d1e015dee0a3acfc97b20a0fa0ff851b03d79ca00df59ce018a63041468\""
						
						str_authorization:=concat('Digest username="admin", realm="',sRealm);
						str_authorization:=concat(str_authorization,'", nonce="');
						str_authorization:=concat(str_authorization,snonce);
						str_authorization:=concat(str_authorization,'", algorithm="SHA-256", uri="/rpc/Switch.GetStatus?id=0", qop=auth, nc=00000001, cnonce="');
						str_authorization:=concat(str_authorization,scnonce);
						str_authorization:=concat(str_authorization,'", response="');
						str_authorization:=concat(str_authorization,str_response);
						str_authorization:=concat(str_authorization,'"');
						
						fbHeader.AddField('Authorization', str_authorization, FALSE);
						IF fbRequest2.SendRequest(sUri:= '/rpc/Switch.GetStatus?id=0', fbClient:= fbClient, eRequestType:= ETcIotHttpRequestType.HTTP_Get, 0, 0, fbHeader) THEN
							nState:= 2;
							bBusy:= TRUE;
							bError:= FALSE;
						END_IF
				END_IF
			END_IF
		END_IF
	
	2:
		IF NOT fbRequest2.bBusy THEN
			bError:= TRUE;
			
			IF NOT fbRequest2.bError THEN				 
				bGetContentResult:= fbRequest2.GetContent(pContent:= ADR(sfincontent), nContentSize:= SIZEOF(sfincontent), bSetNullTermination:= TRUE);
	
				IF fbRequest2.nStatusCode >= 200 AND fbRequest2.nStatusCode < 300 THEN
					bGetJsonResult:= FALSE;
					jsonDoc:= fbRequest2.GetJsonDomContent(fbJson);
					IF jsonDoc <> 0 THEN
						bGetJsonResult:= TRUE;
						IF fbJson.HasMember(jsonDoc, 'output')  THEN
							jsonVal:= fbJson.FindMember(jsonDoc, 'output');
							nValidResCount:= nValidResCount+1;					
							IF fbJson.IsBool(jsonVal) AND (fbJson.GetBool(jsonVal)=TRUE OR fbJson.GetBool(jsonVal)=FALSE) THEN							
								bStateP1:= fbJson.GetBool(jsonVal);									
							END_IF
						END_IF
						IF fbJson.HasMember(jsonDoc, 'apower')  THEN
							jsonVal:= fbJson.FindMember(jsonDoc, 'apower');
							nValidResCount:= nValidResCount+1;
							IF fbJson.IsDouble(jsonVal) AND fbJson.GetDouble(jsonVal)> -3.402823E+38 AND fbJson.GetDouble(jsonVal)< 3.402823E+38 THEN							
								lrapowerP1:= fbJson.GetDouble(jsonVal);									
							END_IF
						END_IF
						IF fbJson.HasMember(jsonDoc, 'voltage')  THEN
							jsonVal:= fbJson.FindMember(jsonDoc, 'voltage');
							nValidResCount:= nValidResCount+1;					
							IF fbJson.IsDouble(jsonVal) AND fbJson.GetDouble(jsonVal)> -3.402823E+38 AND fbJson.GetDouble(jsonVal)< 3.402823E+38 THEN
								lrvoltageP1:= fbJson.GetDouble(jsonVal);									
							END_IF
						END_IF
						IF fbJson.HasMember(jsonDoc, 'temperature')  THEN
							jsonVal:= fbJson.FindMember(jsonDoc, 'temperature');
							 IF fbJson.HasMember(jsonVal, 'tC') AND fbJson.GetDouble(jsonVal)> -3.402823E+38 AND fbJson.GetDouble(jsonVal)< 3.402823E+38 THEN							
								jsonVal:= fbJson.FindMember(jsonVal, 'tC');
								nValidResCount:= nValidResCount+1;					
								IF fbJson.IsDouble(jsonVal) AND fbJson.GetDouble(jsonVal)> -3.402823E+38 AND fbJson.GetDouble(jsonVal)< 3.402823E+38 THEN
									lrTemperatureP1:= fbJson.GetDouble(jsonVal);									
								END_IF
							END_IF
						END_IF
						IF fbJson.HasMember(jsonDoc, 'aenergy')  THEN
							jsonVal:= fbJson.FindMember(jsonDoc, 'aenergy');
							IF fbJson.HasMember(jsonVal, 'total') AND fbJson.GetDouble(jsonVal)> -3.402823E+38 AND fbJson.GetDouble(jsonVal)< 3.402823E+38 THEN							
								jsonVal:= fbJson.FindMember(jsonVal, 'total');
								nValidResCount:= nValidResCount+1;
								IF fbJson.IsDouble(jsonVal) AND fbJson.GetDouble(jsonVal)> -3.402823E+38 AND fbJson.GetDouble(jsonVal)< 3.402823E+38 THEN
									lraenergyP1:= fbJson.GetDouble(jsonVal);
								END_IF
							bError:= FALSE;
							END_IF
						END_IF	
					nResCount:= nResCount+1;			
					END_IF
				END_IF
			END_IF
			
		nState:= 3;
//		bBusy:= FALSE;
			IF bError THEN
				nErrCount:= nErrCount+1;
			END_IF
		END_IF
	
	
	3:
//	IF RisingEdge.Q THEN 
	IF bSetOffP1 AND bStateP1 THEN
		IF fbRequestSwitch1.SendRequest(sUri:= '/rpc/Switch.Set?id=0&on=FALSE', fbClient:= fbClient, eRequestType:= ETcIotHttpRequestType.HTTP_Get, 0, 0, 0) THEN
			nState:= 4;
				nReqCount:= nReqCount+1;
				bBusy:= TRUE;
				bError:= FALSE;
		END_IF
	ELSE
		bBusy:= FALSE;
		bError:= FALSE;
		nState:= 0;
	END_IF	
//	END_IF

		
	4:
		IF NOT fbRequestSwitch1.bBusy THEN
			bError:= TRUE;
			IF NOT fbRequestSwitch1.bError THEN
				bGetContentResult:= fbRequestSwitch1.GetHeaderField(pValue:= ADR(sContentS0), 
														 nValueSize:= SIZEOF(sContentS0), sField := 'WWW-Authenticate');
				IF fbRequestSwitch1.nStatusCode = 401 THEN
					bGetJsonResult:= FALSE;
						sRealm := sContentS0;
						sRealm := DELETE(sRealm, FIND(sRealm, 'realm') + 7, 0);
						sRealm := DELETE(sRealm, LEN(sRealm), FIND(sRealm, '"'));
						
						snonce := sContentS0;
						snonce := DELETE(snonce, FIND(snonce, 'nonce') + 7, 0);
						snonce := DELETE(snonce, LEN(snonce), FIND(snonce, '"'));
						
						scnonce := 'YmawvYzT';
					
						aData := sRealm;
						
						str_Toha1:=concat('admin:', sRealm);
						str_Toha1:=concat(str_Toha1, sPassword);
		 
						udint_length_string:= len2(ADR(str_Toha1));
						F_GenerateHashValue(E_HashMode.HASH_SHA256,ADR(str_Toha1),udint_length_string,ADR(a_ha1),32);
						
							str_ha1:=concat(byte_to_hexstr(a_ha1[0],2,TRUE),byte_to_hexstr(a_ha1[1],2,TRUE));
							str_ha1:=concat(str_ha1,byte_to_hexstr(a_ha1[2],2,TRUE));
							str_ha1:=concat(str_ha1,byte_to_hexstr(a_ha1[3],2,TRUE));
							str_ha1:=concat(str_ha1,byte_to_hexstr(a_ha1[4],2,TRUE));
							str_ha1:=concat(str_ha1,byte_to_hexstr(a_ha1[5],2,TRUE));
							str_ha1:=concat(str_ha1,byte_to_hexstr(a_ha1[6],2,TRUE));
							str_ha1:=concat(str_ha1,byte_to_hexstr(a_ha1[7],2,TRUE));
							str_ha1:=concat(str_ha1,byte_to_hexstr(a_ha1[8],2,TRUE));
							str_ha1:=concat(str_ha1,byte_to_hexstr(a_ha1[9],2,TRUE));
							str_ha1:=concat(str_ha1,byte_to_hexstr(a_ha1[10],2,TRUE));
							str_ha1:=concat(str_ha1,byte_to_hexstr(a_ha1[11],2,TRUE));
							str_ha1:=concat(str_ha1,byte_to_hexstr(a_ha1[12],2,TRUE));
							str_ha1:=concat(str_ha1,byte_to_hexstr(a_ha1[13],2,TRUE));
							str_ha1:=concat(str_ha1,byte_to_hexstr(a_ha1[14],2,TRUE));
							str_ha1:=concat(str_ha1,byte_to_hexstr(a_ha1[15],2,TRUE));
							str_ha1:=concat(str_ha1,byte_to_hexstr(a_ha1[16],2,TRUE));
							str_ha1:=concat(str_ha1,byte_to_hexstr(a_ha1[17],2,TRUE));
							str_ha1:=concat(str_ha1,byte_to_hexstr(a_ha1[18],2,TRUE));
							str_ha1:=concat(str_ha1,byte_to_hexstr(a_ha1[19],2,TRUE));
							str_ha1:=concat(str_ha1,byte_to_hexstr(a_ha1[20],2,TRUE));
							str_ha1:=concat(str_ha1,byte_to_hexstr(a_ha1[21],2,TRUE));
							str_ha1:=concat(str_ha1,byte_to_hexstr(a_ha1[22],2,TRUE));
							str_ha1:=concat(str_ha1,byte_to_hexstr(a_ha1[23],2,TRUE));
							str_ha1:=concat(str_ha1,byte_to_hexstr(a_ha1[24],2,TRUE));
							str_ha1:=concat(str_ha1,byte_to_hexstr(a_ha1[25],2,TRUE));
							str_ha1:=concat(str_ha1,byte_to_hexstr(a_ha1[26],2,TRUE));
							str_ha1:=concat(str_ha1,byte_to_hexstr(a_ha1[27],2,TRUE));
							str_ha1:=concat(str_ha1,byte_to_hexstr(a_ha1[28],2,TRUE));
							str_ha1:=concat(str_ha1,byte_to_hexstr(a_ha1[29],2,TRUE));
							str_ha1:=concat(str_ha1,byte_to_hexstr(a_ha1[30],2,TRUE));
							str_ha1:=concat(str_ha1,byte_to_hexstr(a_ha1[31],2,TRUE));
						
						//str_Toha2:='GET:/rpc/Switch.GetStatus?id=0';
						str_Toha2:='GET:/rpc/Switch.Set?id=0&on=FALSE';
													
						udint_length_string:= len2(ADR(str_Toha2));
						F_GenerateHashValue(E_HashMode.HASH_SHA256,ADR(str_Toha2),udint_length_string,ADR(a_ha2),32);
						
							str_ha2:=concat(byte_to_hexstr(a_ha2[0],2,TRUE),byte_to_hexstr(a_ha2[1],2,TRUE));
							str_ha2:=concat(str_ha2,byte_to_hexstr(a_ha2[2],2,TRUE));
							str_ha2:=concat(str_ha2,byte_to_hexstr(a_ha2[3],2,TRUE));
							str_ha2:=concat(str_ha2,byte_to_hexstr(a_ha2[4],2,TRUE));
							str_ha2:=concat(str_ha2,byte_to_hexstr(a_ha2[5],2,TRUE));
							str_ha2:=concat(str_ha2,byte_to_hexstr(a_ha2[6],2,TRUE));
							str_ha2:=concat(str_ha2,byte_to_hexstr(a_ha2[7],2,TRUE));
							str_ha2:=concat(str_ha2,byte_to_hexstr(a_ha2[8],2,TRUE));
							str_ha2:=concat(str_ha2,byte_to_hexstr(a_ha2[9],2,TRUE));
							str_ha2:=concat(str_ha2,byte_to_hexstr(a_ha2[10],2,TRUE));
							str_ha2:=concat(str_ha2,byte_to_hexstr(a_ha2[11],2,TRUE));
							str_ha2:=concat(str_ha2,byte_to_hexstr(a_ha2[12],2,TRUE));
							str_ha2:=concat(str_ha2,byte_to_hexstr(a_ha2[13],2,TRUE));
							str_ha2:=concat(str_ha2,byte_to_hexstr(a_ha2[14],2,TRUE));
							str_ha2:=concat(str_ha2,byte_to_hexstr(a_ha2[15],2,TRUE));
							str_ha2:=concat(str_ha2,byte_to_hexstr(a_ha2[16],2,TRUE));
							str_ha2:=concat(str_ha2,byte_to_hexstr(a_ha2[17],2,TRUE));
							str_ha2:=concat(str_ha2,byte_to_hexstr(a_ha2[18],2,TRUE));
							str_ha2:=concat(str_ha2,byte_to_hexstr(a_ha2[19],2,TRUE));
							str_ha2:=concat(str_ha2,byte_to_hexstr(a_ha2[20],2,TRUE));
							str_ha2:=concat(str_ha2,byte_to_hexstr(a_ha2[21],2,TRUE));
							str_ha2:=concat(str_ha2,byte_to_hexstr(a_ha2[22],2,TRUE));
							str_ha2:=concat(str_ha2,byte_to_hexstr(a_ha2[23],2,TRUE));
							str_ha2:=concat(str_ha2,byte_to_hexstr(a_ha2[24],2,TRUE));
							str_ha2:=concat(str_ha2,byte_to_hexstr(a_ha2[25],2,TRUE));
							str_ha2:=concat(str_ha2,byte_to_hexstr(a_ha2[26],2,TRUE));
							str_ha2:=concat(str_ha2,byte_to_hexstr(a_ha2[27],2,TRUE));
							str_ha2:=concat(str_ha2,byte_to_hexstr(a_ha2[28],2,TRUE));
							str_ha2:=concat(str_ha2,byte_to_hexstr(a_ha2[29],2,TRUE));
							str_ha2:=concat(str_ha2,byte_to_hexstr(a_ha2[30],2,TRUE));
							str_ha2:=concat(str_ha2,byte_to_hexstr(a_ha2[31],2,TRUE));
							
						// <ha1> + ":" + <nonce> + ":" + <nc> + ":" + <cnonce> + ":" + "auth" + ":" + <ha2>
						
						str_Toresponse:=concat(str_ha1,':');
						str_Toresponse:=concat(str_Toresponse,snonce);
						str_Toresponse:=concat(str_Toresponse,':00000001:');
						str_Toresponse:=concat(str_Toresponse,scnonce);
						str_Toresponse:=concat(str_Toresponse,':');
						str_Toresponse:=concat(str_Toresponse,'auth:');
						str_Toresponse:=concat(str_Toresponse,str_ha2);
						
						udint_length_string:= len2(ADR(str_Toresponse));
						F_GenerateHashValue(E_HashMode.HASH_SHA256,ADR(str_Toresponse),udint_length_string,ADR(a_response),32);
						
